LIN {X 0,Y 323.143,Z 396.929,A -85,B 0,C 180,E1 -15592.369,E2 -15592.369} C_VEL
LIN {X 0,Y 324.214,Z 384.488,A -85,B 0,C 180,E1 -15593.048,E2 -15593.048} C_VEL
LIN {X 0,Y 325.12,Z 370.663,A -85,B 0,C 180,E1 -15593.528,E2 -15593.528} C_VEL
LIN {X 0,Y 327.107,Z 306.154,A -85,B 0,C 180,E1 -15595.157,E2 -15595.157} C_VEL
LIN {X 0,Y 324.289,Z 289.299,A -85,B 0,C 180,E1 -15595.94,E2 -15595.94} C_VEL
LIN {X 0,Y 321.58,Z 277.548,A -85,B 0,C 180,E1 -15596.587,E2 -15596.587} C_VEL
LIN {X 0,Y 317.102,Z 267.049,A -85,B 0,C 180,E1 -15597.471,E2 -15597.471} C_VEL
LIN {X 0,Y 314.783,Z 256.674,A -85,B 0,C 180,E1 -15600.895,E2 -15600.895} C_VEL
LIN {X 0,Y 312.586,Z 248.4,A -85,B 0,C 180,E1 -15603.879,E2 -15603.879} C_VEL
LIN {X 0,Y 312.52,Z 248.065,A -85,B 0,C 180,E1 -15604.205,E2 -15604.205} C_VEL
LIN {X 0,Y 312.522,Z 248.055,A -85,B 0,C 180,E1 -15607.382,E2 -15607.382} C_VEL
LIN {X 0,Y 312.451,Z 248.063,A -85,B 0,C 180,E1 -15610.712,E2 -15610.712} C_VEL
LIN {X 0,Y 312.459,Z 248.066,A -85,B 0,C 180,E1 -15614.204,E2 -15614.204} C_VEL
LIN {X 0,Y 312.461,Z 248.06,A -85,B 0,C 180,E1 -15617.919,E2 -15617.919} C_VEL
LIN {X 0,Y 312.481,Z 248.06,A -85,B 0,C 180,E1 -15621.918,E2 -15621.918} C_VEL
LIN {X 0,Y 312.534,Z 248.049,A -85,B 0,C 180,E1 -15624.213,E2 -15624.213} C_VEL
LIN {X 0,Y 312.505,Z 248.053,A -85,B 0,C 180,E1 -15627.326,E2 -15627.326} C_VEL
LIN {X 0,Y 312.5,Z 248.058,A -85,B 0,C 180,E1 -15631.288,E2 -15631.288} C_VEL
LIN {X 0,Y 312.547,Z 248.049,A -85,B 0,C 180,E1 -15634.7,E2 -15634.7} C_VEL
LIN {X 0,Y 312.538,Z 248.046,A -85,B 0,C 180,E1 -15637.518,E2 -15637.518} C_VEL
LIN {X 0,Y 312.536,Z 248.051,A -85,B 0,C 180,E1 -15641.643,E2 -15641.643} C_VEL
LIN {X 0,Y 312.645,Z 248.04,A -85,B 0,C 180,E1 -15645.676,E2 -15645.676} C_VEL
LIN {X 0,Y 312.675,Z 248.037,A -85,B 0,C 180,E1 -15649.633,E2 -15649.633} C_VEL
LIN {X 0,Y 312.79,Z 248.021,A -85,B 0,C 180,E1 -15652.244,E2 -15652.244} C_VEL
LIN {X 0,Y 312.681,Z 248.031,A -85,B 0,C 180,E1 -15654.834,E2 -15654.834} C_VEL
LIN {X 0,Y 312.97,Z 248.001,A -85,B 0,C 180,E1 -15658.705,E2 -15658.705} C_VEL
LIN {X 0,Y 312.969,Z 248.002,A -85,B 0,C 180,E1 -15661.278,E2 -15661.278} C_VEL
LIN {X 0,Y 312.689,Z 248.033,A -85,B 0,C 180,E1 -15665.149,E2 -15665.149} C_VEL
LIN {X 0,Y 312.839,Z 248.019,A -85,B 0,C 180,E1 -15667.737,E2 -15667.737} C_VEL
LIN {X 0,Y 312.646,Z 248.042,A -85,B 0,C 180,E1 -15671.663,E2 -15671.663} C_VEL
LIN {X 0,Y 312.692,Z 248.117,A -85,B 0,C 180,E1 -15674.304,E2 -15674.304} C_VEL
LIN {X 0,Y 313.537,Z 251.516,A -85,B 0,C 180,E1 -15675.594,E2 -15675.594} C_VEL
LIN {X 0,Y 315.675,Z 259.924,A -85,B 0,C 180,E1 -15678.403,E2 -15678.403} C_VEL
LIN {X 0,Y 322.231,Z 274.036,A -85,B 0,C 180,E1 -15679.641,E2 -15679.641} C_VEL
LIN {X 0,Y 324.868,Z 280.655,A -85,B 0,C 180,E1 -15680.127,E2 -15680.127} C_VEL
LIN {X 0,Y 327.477,Z 294.554,A -85,B 0,C 180,E1 -15680.804,E2 -15680.804} C_VEL
LIN {X 0,Y 324.906,Z 368.524,A -85,B 0,C 180,E1 -15682.683,E2 -15682.683} C_VEL
LIN {X 0,Y 323.933,Z 382.296,A -85,B 0,C 180,E1 -15683.282,E2 -15683.282} C_VEL
LIN {X 0,Y 322.856,Z 394.211,A -85,B 0,C 180,E1 -15684.043,E2 -15684.043} C_VEL
LIN {X 0,Y 321.445,Z 406.032,A -85,B 0,C 180,E1 -15685.052,E2 -15685.052} C_VEL
LIN {X 0,Y 319.906,Z 416.817,A -85,B 0,C 180,E1 -15686.228,E2 -15686.228} C_VEL
LIN {X 0,Y 318.283,Z 427.014,A -85,B 0,C 180,E1 -15687.615,E2 -15687.615} C_VEL
LIN {X 0,Y 316.651,Z 436.505,A -85,B 0,C 180,E1 -15689.216,E2 -15689.216} C_VEL
LIN {X 0,Y 315.049,Z 445.372,A -85,B 0,C 180,E1 -15691.091,E2 -15691.091} C_VEL
LIN {X 0,Y 313.552,Z 453.218,A -85,B 0,C 180,E1 -15693.171,E2 -15693.171} C_VEL
LIN {X 0,Y 312.402,Z 459.627,A -85,B 0,C 180,E1 -15695.387,E2 -15695.387} C_VEL
LIN {X 0,Y 311.579,Z 464.294,A -85,B 0,C 180,E1 -15697.504,E2 -15697.504} C_VEL
LIN {X 0,Y 310.961,Z 467.929,A -85,B 0,C 180,E1 -15699.791,E2 -15699.791} C_VEL
LIN {X 0,Y 310.639,Z 469.904,A -85,B 0,C 180,E1 -15701.707,E2 -15701.707} C_VEL
LIN {X 0,Y 310.454,Z 470.97,A -85,B 0,C 180,E1 -15703.584,E2 -15703.584} C_VEL
LIN {X 0,Y 310.354,Z 471.2,A -85,B 0,C 180,E1 -15705.416,E2 -15705.416} C_VEL
LIN {X 0,Y 310.336,Z 470.655,A -85,B 0,C 180,E1 -15707.208,E2 -15707.208} C_VEL
LIN {X 0,Y 310.409,Z 469.328,A -85,B 0,C 180,E1 -15708.963,E2 -15708.963} C_VEL
LIN {X 0,Y 310.647,Z 467.257,A -85,B 0,C 180,E1 -15710.697,E2 -15710.697} C_VEL
LIN {X 0,Y 310.884,Z 464.494,A -85,B 0,C 180,E1 -15712.387,E2 -15712.387} C_VEL
LIN {X 0,Y 311.332,Z 460.269,A -85,B 0,C 180,E1 -15714.337,E2 -15714.337} C_VEL
LIN {X 0,Y 311.974,Z 454.336,A -85,B 0,C 180,E1 -15716.44,E2 -15716.44} C_VEL
LIN {X 0,Y 312.718,Z 447.541,A -85,B 0,C 180,E1 -15718.348,E2 -15718.348} C_VEL
LIN {X 0,Y 313.675,Z 439.821,A -85,B 0,C 180,E1 -15720.101,E2 -15720.101} C_VEL
LIN {X 0,Y 314.849,Z 430.134,A -85,B 0,C 180,E1 -15721.868,E2 -15721.868} C_VEL
LIN {X 0,Y 316.135,Z 419.363,A -85,B 0,C 180,E1 -15723.441,E2 -15723.441} C_VEL
LIN {X 0,Y 317.364,Z 407.822,A -85,B 0,C 180,E1 -15724.771,E2 -15724.771} C_VEL
LIN {X 0,Y 318.552,Z 394.945,A -85,B 0,C 180,E1 -15725.914,E2 -15725.914} C_VEL
LIN {X 0,Y 319.425,Z 382.214,A -85,B 0,C 180,E1 -15726.748,E2 -15726.748} C_VEL
LIN {X 0,Y 320.216,Z 368.151,A -85,B 0,C 180,E1 -15727.364,E2 -15727.364} C_VEL
LIN {X 0,Y 322.173,Z 291.979,A -85,B 0,C 180,E1 -15729.253,E2 -15729.253} C_VEL
LIN {X 0,Y 318.072,Z 269.596,A -85,B 0,C 180,E1 -15730.109,E2 -15730.109} C_VEL
LIN {X 0,Y 315.028,Z 260.599,A -85,B 0,C 180,E1 -15730.579,E2 -15730.579} C_VEL
LIN {X 0,Y 314.615,Z 258.571,A -85,B 0,C 180,E1 -15731.103,E2 -15731.103} C_VEL
LIN {X 0,Y 312.6,Z 248.111,A -85,B 0,C 180,E1 -15734.656,E2 -15734.656} C_VEL
LIN {X 0,Y 312.602,Z 248.047,A -85,B 0,C 180,E1 -15738.329,E2 -15738.329} C_VEL
LIN {X 0,Y 312.792,Z 248.021,A -85,B 0,C 180,E1 -15742.255,E2 -15742.255} C_VEL
LIN {X 0,Y 312.655,Z 248.041,A -85,B 0,C 180,E1 -15744.844,E2 -15744.844} C_VEL
LIN {X 0,Y 312.892,Z 248.008,A -85,B 0,C 180,E1 -15747.427,E2 -15747.427} C_VEL
LIN {X 0,Y 313.034,Z 247.988,A -85,B 0,C 180,E1 -15750.002,E2 -15750.002} C_VEL
LIN {X 0,Y 312.893,Z 248.008,A -85,B 0,C 180,E1 -15752.577,E2 -15752.577} C_VEL
LIN {X 0,Y 312.838,Z 248.013,A -85,B 0,C 180,E1 -15756.452,E2 -15756.452} C_VEL
LIN {X 0,Y 312.721,Z 248.031,A -85,B 0,C 180,E1 -15759.053,E2 -15759.053} C_VEL
LIN {X 0,Y 312.57,Z 248.048,A -85,B 0,C 180,E1 -15762.996,E2 -15762.996} C_VEL
LIN {X 0,Y 312.564,Z 248.051,A -85,B 0,C 180,E1 -15765.656,E2 -15765.656} C_VEL
LIN {X 0,Y 312.549,Z 248.047,A -85,B 0,C 180,E1 -15769.23,E2 -15769.23} C_VEL
LIN {X 0,Y 312.47,Z 248.059,A -85,B 0,C 180,E1 -15772.787,E2 -15772.787} C_VEL
LIN {X 0,Y 312.547,Z 248.052,A -85,B 0,C 180,E1 -15775.942,E2 -15775.942} C_VEL
LIN {X 0,Y 312.493,Z 248.051,A -85,B 0,C 180,E1 -15779.657,E2 -15779.657} C_VEL
LIN {X 0,Y 312.471,Z 248.06,A -85,B 0,C 180,E1 -15783.697,E2 -15783.697} C_VEL
LIN {X 0,Y 312.494,Z 248.055,A -85,B 0,C 180,E1 -15787.392,E2 -15787.392} C_VEL
LIN {X 0,Y 312.485,Z 248.06,A -85,B 0,C 180,E1 -15790.712,E2 -15790.712} C_VEL
LIN {X 0,Y 312.556,Z 248.051,A -85,B 0,C 180,E1 -15794.193,E2 -15794.193} C_VEL
LIN {X 0,Y 312.525,Z 248.049,A -85,B 0,C 180,E1 -15794.965,E2 -15794.965} C_VEL
LIN {X 0,Y 311.856,Z 248.137,A -85,B 0,C 180,E1 -15796.041,E2 -15796.041} C_VEL
LIN {X 0,Y 308.981,Z 248.492,A -85,B 0,C 180,E1 -15797.79,E2 -15797.79} C_VEL
LIN {X 0,Y 306.546,Z 248.798,A -85,B 0,C 180,E1 -15799.209,E2 -15799.209} C_VEL
LIN {X 0,Y 305.509,Z 248.928,A -85,B 0,C 180,E1 -15800.309,E2 -15800.309} C_VEL
LIN {X 0,Y 305.43,Z 248.932,A -85,B 0,C 180,E1 -15800.681,E2 -15800.681} C_VEL
LIN {X 0,Y 305.474,Z 248.929,A -85,B 0,C 180,E1 -15803.636,E2 -15803.636} C_VEL
LIN {X 0,Y 305.439,Z 248.934,A -85,B 0,C 180,E1 -15806.493,E2 -15806.493} C_VEL
LIN {X 0,Y 305.435,Z 248.936,A -85,B 0,C 180,E1 -15809.6,E2 -15809.6} C_VEL
LIN {X 0,Y 305.476,Z 248.931,A -85,B 0,C 180,E1 -15812.616,E2 -15812.616} C_VEL
LIN {X 0,Y 305.488,Z 248.93,A -85,B 0,C 180,E1 -15815.548,E2 -15815.548} C_VEL
LIN {X 0,Y 305.471,Z 248.932,A -85,B 0,C 180,E1 -15819.822,E2 -15819.822} C_VEL
LIN {X 0,Y 305.543,Z 248.921,A -85,B 0,C 180,E1 -15823.987,E2 -15823.987} C_VEL
LIN {X 0,Y 305.582,Z 248.916,A -85,B 0,C 180,E1 -15826.714,E2 -15826.714} C_VEL
LIN {X 0,Y 305.753,Z 248.896,A -85,B 0,C 180,E1 -15831.271,E2 -15831.271} C_VEL
LIN {X 0,Y 305.788,Z 248.89,A -85,B 0,C 180,E1 -15833.41,E2 -15833.41} C_VEL
LIN {X 0,Y 305.866,Z 248.883,A -85,B 0,C 180,E1 -15837.375,E2 -15837.375} C_VEL
LIN {X 0,Y 305.923,Z 248.879,A -85,B 0,C 180,E1 -15840.009,E2 -15840.009} C_VEL
LIN {X 0,Y 305.862,Z 248.878,A -85,B 0,C 180,E1 -15842.642,E2 -15842.642} C_VEL
LIN {X 0,Y 305.798,Z 248.887,A -85,B 0,C 180,E1 -15846.607,E2 -15846.607} C_VEL
LIN {X 0,Y 305.708,Z 248.899,A -85,B 0,C 180,E1 -15849.269,E2 -15849.269} C_VEL
LIN {X 0,Y 305.602,Z 248.915,A -85,B 0,C 180,E1 -15853.303,E2 -15853.303} C_VEL
LIN {X 0,Y 305.569,Z 248.918,A -85,B 0,C 180,E1 -15856.029,E2 -15856.029} C_VEL
LIN {X 0,Y 305.502,Z 248.923,A -85,B 0,C 180,E1 -15860.194,E2 -15860.194} C_VEL
LIN {X 0,Y 305.509,Z 248.93,A -85,B 0,C 180,E1 -15863.045,E2 -15863.045} C_VEL
LIN {X 0,Y 305.49,Z 248.928,A -85,B 0,C 180,E1 -15866.201,E2 -15866.201} C_VEL
LIN {X 0,Y 305.458,Z 248.933,A -85,B 0,C 180,E1 -15869.034,E2 -15869.034} C_VEL
LIN {X 0,Y 305.461,Z 248.932,A -85,B 0,C 180,E1 -15871.958,E2 -15871.958} C_VEL
LIN {X 0,Y 305.487,Z 248.933,A -85,B 0,C 180,E1 -15875.118,E2 -15875.118} C_VEL
LIN {X 0,Y 305.46,Z 248.932,A -85,B 0,C 180,E1 -15878.529,E2 -15878.529} C_VEL
LIN {X 0,Y 305.405,Z 248.937,A -85,B 0,C 180,E1 -15882.573,E2 -15882.573} C_VEL
LIN {X 0,Y 305.408,Z 248.938,A -85,B 0,C 180,E1 -15886.339,E2 -15886.339} C_VEL
LIN {X 0,Y 305.418,Z 248.942,A -85,B 0,C 180,E1 -15889.884,E2 -15889.884} C_VEL
LIN {X 0,Y 305.487,Z 248.934,A -85,B 0,C 180,E1 -15893.639,E2 -15893.639} C_VEL
LIN {X 0,Y 305.492,Z 248.931,A -85,B 0,C 180,E1 -15896.484,E2 -15896.484} C_VEL
LIN {X 0,Y 305.517,Z 249.096,A -85,B 0,C 180,E1 -15898.924,E2 -15898.924} C_VEL
LIN {X 0,Y 307.752,Z 259.847,A -85,B 0,C 180,E1 -15902.453,E2 -15902.453} C_VEL
LIN {X 0,Y 309.311,Z 268.287,A -85,B 0,C 180,E1 -15905.027,E2 -15905.027} C_VEL
LIN {X 0,Y 310.261,Z 273.009,A -85,B 0,C 180,E1 -15905.272,E2 -15905.272} C_VEL
LIN {X 0,Y 315.347,Z 307.012,A -85,B 0,C 180,E1 -15906.527,E2 -15906.527} C_VEL
LIN {X 0,Y 313.49,Z 375.371,A -85,B 0,C 180,E1 -15908.245,E2 -15908.245} C_VEL
LIN {X 0,Y 312.701,Z 389.193,A -85,B 0,C 180,E1 -15908.836,E2 -15908.836} C_VEL
LIN {X 0,Y 311.73,Z 401.738,A -85,B 0,C 180,E1 -15909.63,E2 -15909.63} C_VEL
LIN {X 0,Y 310.555,Z 413.817,A -85,B 0,C 180,E1 -15910.67,E2 -15910.67} C_VEL
LIN {X 0,Y 309.233,Z 425.375,A -85,B 0,C 180,E1 -15911.959,E2 -15911.959} C_VEL
LIN {X 0,Y 308.113,Z 435.341,A -85,B 0,C 180,E1 -15913.354,E2 -15913.354} C_VEL
LIN {X 0,Y 306.849,Z 445.2,A -85,B 0,C 180,E1 -15915.066,E2 -15915.066} C_VEL
LIN {X 0,Y 305.701,Z 454.297,A -85,B 0,C 180,E1 -15917.045,E2 -15917.045} C_VEL
LIN {X 0,Y 304.831,Z 461.601,A -85,B 0,C 180,E1 -15919.033,E2 -15919.033} C_VEL
LIN {X 0,Y 304.321,Z 466.519,A -85,B 0,C 180,E1 -15920.695,E2 -15920.695} C_VEL
LIN {X 0,Y 303.879,Z 471.271,A -85,B 0,C 180,E1 -15922.69,E2 -15922.69} C_VEL
LIN {X 0,Y 303.663,Z 474.872,A -85,B 0,C 180,E1 -15924.686,E2 -15924.686} C_VEL
LIN {X 0,Y 303.6,Z 476.688,A -85,B 0,C 180,E1 -15926.016,E2 -15926.016} C_VEL
LIN {X 0,Y 303.592,Z 478.049,A -85,B 0,C 180,E1 -15927.344,E2 -15927.344} C_VEL
LIN {X 0,Y 303.54,Z 479.001,A -85,B 0,C 180,E1 -15928.671,E2 -15928.671} C_VEL
LIN {X 0,Y 303.547,Z 479.553,A -85,B 0,C 180,E1 -15929.998,E2 -15929.998} C_VEL
LIN {X 0,Y 303.539,Z 479.658,A -85,B 0,C 180,E1 -15931.324,E2 -15931.324} C_VEL
LIN {X 0,Y 303.592,Z 479.358,A -85,B 0,C 180,E1 -15932.651,E2 -15932.651} C_VEL
LIN {X 0,Y 303.606,Z 478.665,A -85,B 0,C 180,E1 -15933.98,E2 -15933.98} C_VEL
LIN {X 0,Y 303.718,Z 477.175,A -85,B 0,C 180,E1 -15935.676,E2 -15935.676} C_VEL
LIN {X 0,Y 304.09,Z 474.055,A -85,B 0,C 180,E1 -15937.968,E2 -15937.968} C_VEL
LIN {X 0,Y 304.709,Z 470.241,A -85,B 0,C 180,E1 -15939.959,E2 -15939.959} C_VEL
LIN {X 0,Y 305.562,Z 465.301,A -85,B 0,C 180,E1 -15941.944,E2 -15941.944} C_VEL
LIN {X 0,Y 306.698,Z 459.092,A -85,B 0,C 180,E1 -15943.92,E2 -15943.92} C_VEL
LIN {X 0,Y 308.341,Z 451.381,A -85,B 0,C 180,E1 -15945.871,E2 -15945.871} C_VEL
LIN {X 0,Y 310.033,Z 441.588,A -85,B 0,C 180,E1 -15947.851,E2 -15947.851} C_VEL
LIN {X 0,Y 311.728,Z 431.881,A -85,B 0,C 180,E1 -15949.421,E2 -15949.421} C_VEL
LIN {X 0,Y 313.597,Z 420.806,A -85,B 0,C 180,E1 -15950.838,E2 -15950.838} C_VEL
LIN {X 0,Y 315.366,Z 408.317,A -85,B 0,C 180,E1 -15952.087,E2 -15952.087} C_VEL
LIN {X 0,Y 316.922,Z 396.004,A -85,B 0,C 180,E1 -15953.005,E2 -15953.005} C_VEL
LIN {X 0,Y 318.017,Z 383.244,A -85,B 0,C 180,E1 -15953.696,E2 -15953.696} C_VEL
LIN {X 0,Y 318.88,Z 370.165,A -85,B 0,C 180,E1 -15954.146,E2 -15954.146} C_VEL
LIN {X 0,Y 320.97,Z 307.114,A -85,B 0,C 180,E1 -15955.769,E2 -15955.769} C_VEL
LIN {X 0,Y 318.251,Z 290.858,A -85,B 0,C 180,E1 -15956.562,E2 -15956.562} C_VEL
LIN {X 0,Y 316.086,Z 280.936,A -85,B 0,C 180,E1 -15957.114,E2 -15957.114} C_VEL
LIN {X 0,Y 311.207,Z 269.934,A -85,B 0,C 180,E1 -15958.066,E2 -15958.066} C_VEL
LIN {X 0,Y 309.962,Z 267.008,A -85,B 0,C 180,E1 -15958.344,E2 -15958.344} C_VEL
LIN {X 0,Y 307.674,Z 257.238,A -85,B 0,C 180,E1 -15961.69,E2 -15961.69} C_VEL
LIN {X 0,Y 305.505,Z 249.086,A -85,B 0,C 180,E1 -15964.816,E2 -15964.816} C_VEL
LIN {X 0,Y 305.446,Z 248.939,A -85,B 0,C 180,E1 -15968.519,E2 -15968.519} C_VEL
LIN {X 0,Y 305.444,Z 248.937,A -85,B 0,C 180,E1 -15972.575,E2 -15972.575} C_VEL
LIN {X 0,Y 305.428,Z 248.939,A -85,B 0,C 180,E1 -15976.337,E2 -15976.337} C_VEL
LIN {X 0,Y 305.417,Z 248.94,A -85,B 0,C 180,E1 -15979.878,E2 -15979.878} C_VEL
LIN {X 0,Y 305.466,Z 248.928,A -85,B 0,C 180,E1 -15983.631,E2 -15983.631} C_VEL
LIN {X 0,Y 305.469,Z 248.929,A -85,B 0,C 180,E1 -15986.476,E2 -15986.476} C_VEL
LIN {X 0,Y 305.421,Z 248.936,A -85,B 0,C 180,E1 -15989.579,E2 -15989.579} C_VEL
LIN {X 0,Y 305.455,Z 248.933,A -85,B 0,C 180,E1 -15992.594,E2 -15992.594} C_VEL
LIN {X 0,Y 305.473,Z 248.933,A -85,B 0,C 180,E1 -15995.528,E2 -15995.528} C_VEL
LIN {X 0,Y 305.456,Z 248.933,A -85,B 0,C 180,E1 -15998.392,E2 -15998.392} C_VEL
LIN {X 0,Y 305.495,Z 248.924,A -85,B 0,C 180,E1 -16001.204,E2 -16001.204} C_VEL
LIN {X 0,Y 305.572,Z 248.919,A -85,B 0,C 180,E1 -16005.337,E2 -16005.337} C_VEL
LIN {X 0,Y 305.614,Z 248.918,A -85,B 0,C 180,E1 -16009.391,E2 -16009.391} C_VEL
LIN {X 0,Y 305.74,Z 248.899,A -85,B 0,C 180,E1 -16012.064,E2 -16012.064} C_VEL
LIN {X 0,Y 305.651,Z 248.906,A -85,B 0,C 180,E1 -16014.714,E2 -16014.714} C_VEL
LIN {X 0,Y 305.936,Z 248.877,A -85,B 0,C 180,E1 -16018.675,E2 -16018.675} C_VEL
LIN {X 0,Y 305.936,Z 248.879,A -85,B 0,C 180,E1 -16021.308,E2 -16021.308} C_VEL
LIN {X 0,Y 305.661,Z 248.909,A -85,B 0,C 180,E1 -16025.268,E2 -16025.268} C_VEL
LIN {X 0,Y 305.782,Z 248.898,A -85,B 0,C 180,E1 -16027.917,E2 -16027.917} C_VEL
LIN {X 0,Y 305.58,Z 248.921,A -85,B 0,C 180,E1 -16031.936,E2 -16031.936} C_VEL
LIN {X 0,Y 305.601,Z 248.982,A -85,B 0,C 180,E1 -16033.455,E2 -16033.455} C_VEL
LIN {X 0,Y 307.131,Z 254.679,A -85,B 0,C 180,E1 -16035.653,E2 -16035.653} C_VEL
LIN {X 0,Y 308.543,Z 260.196,A -85,B 0,C 180,E1 -16037.522,E2 -16037.522} C_VEL
LIN {X 0,Y 314.968,Z 273.498,A -85,B 0,C 180,E1 -16038.783,E2 -16038.783} C_VEL
LIN {X 0,Y 319.191,Z 283.718,A -85,B 0,C 180,E1 -16039.588,E2 -16039.588} C_VEL
LIN {X 0,Y 321.366,Z 295.811,A -85,B 0,C 180,E1 -16040.196,E2 -16040.196} C_VEL
LIN {X 0,Y 318.671,Z 368.497,A -85,B 0,C 180,E1 -16042.078,E2 -16042.078} C_VEL
LIN {X 0,Y 317.615,Z 382.644,A -85,B 0,C 180,E1 -16042.703,E2 -16042.703} C_VEL
LIN {X 0,Y 316.41,Z 395.453,A -85,B 0,C 180,E1 -16043.555,E2 -16043.555} C_VEL
LIN {X 0,Y 314.75,Z 408.209,A -85,B 0,C 180,E1 -16044.699,E2 -16044.699} C_VEL
LIN {X 0,Y 313.273,Z 417.956,A -85,B 0,C 180,E1 -16045.816,E2 -16045.816} C_VEL
LIN {X 0,Y 311.448,Z 428.762,A -85,B 0,C 180,E1 -16047.361,E2 -16047.361} C_VEL
LIN {X 0,Y 309.732,Z 437.936,A -85,B 0,C 180,E1 -16049.001,E2 -16049.001} C_VEL
LIN {X 0,Y 308.111,Z 446.353,A -85,B 0,C 180,E1 -16050.866,E2 -16050.866} C_VEL
LIN {X 0,Y 306.525,Z 454.18,A -85,B 0,C 180,E1 -16053.056,E2 -16053.056} C_VEL
LIN {X 0,Y 305.429,Z 459.882,A -85,B 0,C 180,E1 -16055.104,E2 -16055.104} C_VEL
LIN {X 0,Y 304.475,Z 465.022,A -85,B 0,C 180,E1 -16057.538,E2 -16057.538} C_VEL
LIN {X 0,Y 303.964,Z 467.842,A -85,B 0,C 180,E1 -16059.404,E2 -16059.404} C_VEL
LIN {X 0,Y 303.745,Z 468.961,A -85,B 0,C 180,E1 -16060.366,E2 -16060.366} C_VEL
LIN {X 0,Y 303.483,Z 470.477,A -85,B 0,C 180,E1 -16062.183,E2 -16062.183} C_VEL
LIN {X 0,Y 303.309,Z 471.256,A -85,B 0,C 180,E1 -16064.089,E2 -16064.089} C_VEL
LIN {X 0,Y 303.256,Z 471.21,A -85,B 0,C 180,E1 -16065.956,E2 -16065.956} C_VEL
LIN {X 0,Y 303.261,Z 470.311,A -85,B 0,C 180,E1 -16067.85,E2 -16067.85} C_VEL
LIN {X 0,Y 303.404,Z 468.473,A -85,B 0,C 180,E1 -16069.836,E2 -16069.836} C_VEL
LIN {X 0,Y 303.728,Z 465.6,A -85,B 0,C 180,E1 -16071.862,E2 -16071.862} C_VEL
LIN {X 0,Y 304.141,Z 461.488,A -85,B 0,C 180,E1 -16073.955,E2 -16073.955} C_VEL
LIN {X 0,Y 304.736,Z 455.931,A -85,B 0,C 180,E1 -16076.103,E2 -16076.103} C_VEL
LIN {X 0,Y 305.6,Z 448.588,A -85,B 0,C 180,E1 -16078.287,E2 -16078.287} C_VEL
LIN {X 0,Y 306.581,Z 440.79,A -85,B 0,C 180,E1 -16080.14,E2 -16080.14} C_VEL
LIN {X 0,Y 307.725,Z 431.805,A -85,B 0,C 180,E1 -16081.872,E2 -16081.872} C_VEL
LIN {X 0,Y 309.047,Z 421.239,A -85,B 0,C 180,E1 -16083.497,E2 -16083.497} C_VEL
LIN {X 0,Y 310.332,Z 409.706,A -85,B 0,C 180,E1 -16084.912,E2 -16084.912} C_VEL
LIN {X 0,Y 311.477,Z 397.841,A -85,B 0,C 180,E1 -16086.04,E2 -16086.04} C_VEL
LIN {X 0,Y 312.437,Z 385.507,A -85,B 0,C 180,E1 -16086.928,E2 -16086.928} C_VEL
LIN {X 0,Y 313.255,Z 372.677,A -85,B 0,C 180,E1 -16087.582,E2 -16087.582} C_VEL
LIN {X 0,Y 313.807,Z 357.919,A -85,B 0,C 180,E1 -16088.035,E2 -16088.035} C_VEL
LIN {X 0,Y 315.483,Z 292.998,A -85,B 0,C 180,E1 -16089.654,E2 -16089.654} C_VEL
LIN {X 0,Y 311.694,Z 271.957,A -85,B 0,C 180,E1 -16090.47,E2 -16090.47} C_VEL
LIN {X 0,Y 307.771,Z 260.477,A -85,B 0,C 180,E1 -16091.099,E2 -16091.099} C_VEL
LIN {X 0,Y 306.433,Z 253.556,A -85,B 0,C 180,E1 -16093.343,E2 -16093.343} C_VEL
LIN {X 0,Y 305.603,Z 248.978,A -85,B 0,C 180,E1 -16094.993,E2 -16094.993} C_VEL
LIN {X 0,Y 305.57,Z 248.92,A -85,B 0,C 180,E1 -16099.4,E2 -16099.4} C_VEL
LIN {X 0,Y 305.734,Z 248.899,A -85,B 0,C 180,E1 -16102.075,E2 -16102.075} C_VEL
LIN {X 0,Y 305.625,Z 248.917,A -85,B 0,C 180,E1 -16104.725,E2 -16104.725} C_VEL
LIN {X 0,Y 305.894,Z 248.882,A -85,B 0,C 180,E1 -16108.686,E2 -16108.686} C_VEL
LIN {X 0,Y 305.895,Z 248.882,A -85,B 0,C 180,E1 -16111.319,E2 -16111.319} C_VEL
LIN {X 0,Y 305.627,Z 248.916,A -85,B 0,C 180,E1 -16115.28,E2 -16115.28} C_VEL
LIN {X 0,Y 305.738,Z 248.898,A -85,B 0,C 180,E1 -16117.93,E2 -16117.93} C_VEL
LIN {X 0,Y 305.54,Z 248.923,A -85,B 0,C 180,E1 -16121.95,E2 -16121.95} C_VEL
LIN {X 0,Y 305.558,Z 248.922,A -85,B 0,C 180,E1 -16125.027,E2 -16125.027} C_VEL
LIN {X 0,Y 305.519,Z 248.92,A -85,B 0,C 180,E1 -16128.789,E2 -16128.789} C_VEL
LIN {X 0,Y 305.43,Z 248.936,A -85,B 0,C 180,E1 -16133.046,E2 -16133.046} C_VEL
LIN {X 0,Y 305.477,Z 248.929,A -85,B 0,C 180,E1 -16136.228,E2 -16136.228} C_VEL
LIN {X 0,Y 305.442,Z 248.926,A -85,B 0,C 180,E1 -16139.057,E2 -16139.057} C_VEL
LIN {X 0,Y 305.397,Z 248.941,A -85,B 0,C 180,E1 -16141.96,E2 -16141.96} C_VEL
LIN {X 0,Y 305.414,Z 248.938,A -85,B 0,C 180,E1 -16145.122,E2 -16145.122} C_VEL
LIN {X 0,Y 305.438,Z 248.937,A -85,B 0,C 180,E1 -16148.545,E2 -16148.545} C_VEL
LIN {X 0,Y 305.481,Z 248.934,A -85,B 0,C 180,E1 -16152.608,E2 -16152.608} C_VEL
LIN {X 0,Y 305.497,Z 248.93,A -85,B 0,C 180,E1 -16156.374,E2 -16156.374} C_VEL
LIN {X 0,Y 305.453,Z 248.933,A -85,B 0,C 180,E1 -16159.906,E2 -16159.906} C_VEL
LIN {X 0,Y 305.43,Z 248.932,A -85,B 0,C 180,E1 -16160.681,E2 -16160.681} C_VEL
LIN {X 0,Y 304.768,Z 249.019,A -85,B 0,C 180,E1 -16161.781,E2 -16161.781} C_VEL
LIN {X 0,Y 301.899,Z 249.374,A -85,B 0,C 180,E1 -16163.572,E2 -16163.572} C_VEL
LIN {X 0,Y 299.464,Z 249.68,A -85,B 0,C 180,E1 -16165.025,E2 -16165.025} C_VEL
LIN {X 0,Y 298.426,Z 249.805,A -85,B 0,C 180,E1 -16166.15,E2 -16166.15} C_VEL
LIN {X 0,Y 298.346,Z 249.815,A -85,B 0,C 180,E1 -16166.532,E2 -16166.532} C_VEL
LIN {X 0,Y 298.406,Z 249.813,A -85,B 0,C 180,E1 -16170.627,E2 -16170.627} C_VEL
LIN {X 0,Y 298.458,Z 249.803,A -85,B 0,C 180,E1 -16173.488,E2 -16173.488} C_VEL
LIN {X 0,Y 298.416,Z 249.809,A -85,B 0,C 180,E1 -16176.71,E2 -16176.71} C_VEL
LIN {X 0,Y 298.453,Z 249.805,A -85,B 0,C 180,E1 -16180.762,E2 -16180.762} C_VEL
LIN {X 0,Y 298.58,Z 249.787,A -85,B 0,C 180,E1 -16185.004,E2 -16185.004} C_VEL
LIN {X 0,Y 298.589,Z 249.789,A -85,B 0,C 180,E1 -16189.156,E2 -16189.156} C_VEL
LIN {X 0,Y 298.699,Z 249.775,A -85,B 0,C 180,E1 -16191.894,E2 -16191.894} C_VEL
LIN {X 0,Y 298.636,Z 249.781,A -85,B 0,C 180,E1 -16194.608,E2 -16194.608} C_VEL
LIN {X 0,Y 298.91,Z 249.748,A -85,B 0,C 180,E1 -16198.662,E2 -16198.662} C_VEL
LIN {X 0,Y 298.92,Z 249.744,A -85,B 0,C 180,E1 -16201.356,E2 -16201.356} C_VEL
LIN {X 0,Y 298.746,Z 249.763,A -85,B 0,C 180,E1 -16206.763,E2 -16206.763} C_VEL
LIN {X 0,Y 298.639,Z 249.78,A -85,B 0,C 180,E1 -16209.49,E2 -16209.49} C_VEL
LIN {X 0,Y 298.562,Z 249.792,A -85,B 0,C 180,E1 -16213.623,E2 -16213.623} C_VEL
LIN {X 0,Y 298.502,Z 249.801,A -85,B 0,C 180,E1 -16216.419,E2 -16216.419} C_VEL
LIN {X 0,Y 298.465,Z 249.798,A -85,B 0,C 180,E1 -16219.625,E2 -16219.625} C_VEL
LIN {X 0,Y 298.442,Z 249.807,A -85,B 0,C 180,E1 -16223.607,E2 -16223.607} C_VEL
LIN {X 0,Y 298.43,Z 249.81,A -85,B 0,C 180,E1 -16226.588,E2 -16226.588} C_VEL
LIN {X 0,Y 298.385,Z 249.812,A -85,B 0,C 180,E1 -16229.653,E2 -16229.653} C_VEL
LIN {X 0,Y 298.418,Z 249.812,A -85,B 0,C 180,E1 -16232.805,E2 -16232.805} C_VEL
LIN {X 0,Y 298.429,Z 249.804,A -85,B 0,C 180,E1 -16236.076,E2 -16236.076} C_VEL
LIN {X 0,Y 298.399,Z 249.817,A -85,B 0,C 180,E1 -16239.496,E2 -16239.496} C_VEL
LIN {X 0,Y 298.367,Z 249.815,A -85,B 0,C 180,E1 -16243.094,E2 -16243.094} C_VEL
LIN {X 0,Y 298.367,Z 249.814,A -85,B 0,C 180,E1 -16246.912,E2 -16246.912} C_VEL
LIN {X 0,Y 298.389,Z 249.814,A -85,B 0,C 180,E1 -16251.019,E2 -16251.019} C_VEL
LIN {X 0,Y 298.43,Z 249.813,A -85,B 0,C 180,E1 -16253.93,E2 -16253.93} C_VEL
LIN {X 0,Y 298.42,Z 249.812,A -85,B 0,C 180,E1 -16257.201,E2 -16257.201} C_VEL
LIN {X 0,Y 298.466,Z 250.004,A -85,B 0,C 180,E1 -16258.583,E2 -16258.583} C_VEL
LIN {X 0,Y 300.654,Z 260.561,A -85,B 0,C 180,E1 -16262.125,E2 -16262.125} C_VEL
LIN {X 0,Y 302.165,Z 268.328,A -85,B 0,C 180,E1 -16264.541,E2 -16264.541} C_VEL
LIN {X 0,Y 303.685,Z 274.375,A -85,B 0,C 180,E1 -16264.856,E2 -16264.856} C_VEL
LIN {X 0,Y 308.657,Z 307.144,A -85,B 0,C 180,E1 -16266.102,E2 -16266.102} C_VEL
LIN {X 0,Y 306.701,Z 375.684,A -85,B 0,C 180,E1 -16267.871,E2 -16267.871} C_VEL
LIN {X 0,Y 305.879,Z 389.329,A -85,B 0,C 180,E1 -16268.473,E2 -16268.473} C_VEL
LIN {X 0,Y 304.848,Z 402.357,A -85,B 0,C 180,E1 -16269.326,E2 -16269.326} C_VEL
LIN {X 0,Y 303.639,Z 414.234,A -85,B 0,C 180,E1 -16270.388,E2 -16270.388} C_VEL
LIN {X 0,Y 302.281,Z 425.7,A -85,B 0,C 180,E1 -16271.705,E2 -16271.705} C_VEL
LIN {X 0,Y 301.151,Z 435.516,A -85,B 0,C 180,E1 -16273.119,E2 -16273.119} C_VEL
LIN {X 0,Y 299.968,Z 444.552,A -85,B 0,C 180,E1 -16274.715,E2 -16274.715} C_VEL
LIN {X 0,Y 298.753,Z 453.743,A -85,B 0,C 180,E1 -16276.738,E2 -16276.738} C_VEL
LIN {X 0,Y 297.825,Z 461.137,A -85,B 0,C 180,E1 -16278.772,E2 -16278.772} C_VEL
LIN {X 0,Y 297.286,Z 466.118,A -85,B 0,C 180,E1 -16280.472,E2 -16280.472} C_VEL
LIN {X 0,Y 296.828,Z 470.936,A -85,B 0,C 180,E1 -16282.515,E2 -16282.515} C_VEL
LIN {X 0,Y 296.578,Z 474.597,A -85,B 0,C 180,E1 -16284.559,E2 -16284.559} C_VEL
LIN {X 0,Y 296.504,Z 476.467,A -85,B 0,C 180,E1 -16285.92,E2 -16285.92} C_VEL
LIN {X 0,Y 296.497,Z 477.856,A -85,B 0,C 180,E1 -16287.28,E2 -16287.28} C_VEL
LIN {X 0,Y 296.463,Z 478.836,A -85,B 0,C 180,E1 -16288.639,E2 -16288.639} C_VEL
LIN {X 0,Y 296.465,Z 479.417,A -85,B 0,C 180,E1 -16289.998,E2 -16289.998} C_VEL
LIN {X 0,Y 296.461,Z 479.571,A -85,B 0,C 180,E1 -16291.356,E2 -16291.356} C_VEL
LIN {X 0,Y 296.498,Z 479.296,A -85,B 0,C 180,E1 -16292.715,E2 -16292.715} C_VEL
LIN {X 0,Y 296.509,Z 478.628,A -85,B 0,C 180,E1 -16294.075,E2 -16294.075} C_VEL
LIN {X 0,Y 296.604,Z 477.441,A -85,B 0,C 180,E1 -16295.574,E2 -16295.574} C_VEL
LIN {X 0,Y 297.058,Z 474.116,A -85,B 0,C 180,E1 -16298.158,E2 -16298.158} C_VEL
LIN {X 0,Y 297.704,Z 470.353,A -85,B 0,C 180,E1 -16300.196,E2 -16300.196} C_VEL
LIN {X 0,Y 298.614,Z 465.482,A -85,B 0,C 180,E1 -16302.226,E2 -16302.226} C_VEL
LIN {X 0,Y 299.82,Z 459.358,A -85,B 0,C 180,E1 -16304.246,E2 -16304.246} C_VEL
LIN {X 0,Y 301.536,Z 451.753,A -85,B 0,C 180,E1 -16306.239,E2 -16306.239} C_VEL
LIN {X 0,Y 303.128,Z 443.106,A -85,B 0,C 180,E1 -16308.072,E2 -16308.072} C_VEL
LIN {X 0,Y 304.876,Z 433.559,A -85,B 0,C 180,E1 -16309.7,E2 -16309.7} C_VEL
LIN {X 0,Y 306.763,Z 422.953,A -85,B 0,C 180,E1 -16311.149,E2 -16311.149} C_VEL
LIN {X 0,Y 308.392,Z 412.764,A -85,B 0,C 180,E1 -16312.261,E2 -16312.261} C_VEL
LIN {X 0,Y 310.127,Z 400.734,A -85,B 0,C 180,E1 -16313.273,E2 -16313.273} C_VEL
LIN {X 0,Y 311.389,Z 387.754,A -85,B 0,C 180,E1 -16314.1,E2 -16314.1} C_VEL
LIN {X 0,Y 312.449,Z 375.125,A -85,B 0,C 180,E1 -16314.632,E2 -16314.632} C_VEL
LIN {X 0,Y 314.907,Z 308.047,A -85,B 0,C 180,E1 -16316.417,E2 -16316.417} C_VEL
LIN {X 0,Y 312.328,Z 292.521,A -85,B 0,C 180,E1 -16317.202,E2 -16317.202} C_VEL
LIN {X 0,Y 310.387,Z 283.805,A -85,B 0,C 180,E1 -16317.715,E2 -16317.715} C_VEL
LIN {X 0,Y 304.742,Z 270.974,A -85,B 0,C 180,E1 -16318.873,E2 -16318.873} C_VEL
LIN {X 0,Y 302.669,Z 266.657,A -85,B 0,C 180,E1 -16319.355,E2 -16319.355} C_VEL
LIN {X 0,Y 300.513,Z 257.553,A -85,B 0,C 180,E1 -16322.647,E2 -16322.647} C_VEL
LIN {X 0,Y 298.439,Z 249.914,A -85,B 0,C 180,E1 -16325.753,E2 -16325.753} C_VEL
LIN {X 0,Y 298.386,Z 249.815,A -85,B 0,C 180,E1 -16329.486,E2 -16329.486} C_VEL
LIN {X 0,Y 298.379,Z 249.814,A -85,B 0,C 180,E1 -16333.09,E2 -16333.09} C_VEL
LIN {X 0,Y 298.378,Z 249.818,A -85,B 0,C 180,E1 -16336.908,E2 -16336.908} C_VEL
LIN {X 0,Y 298.392,Z 249.811,A -85,B 0,C 180,E1 -16341.004,E2 -16341.004} C_VEL
LIN {X 0,Y 298.408,Z 249.808,A -85,B 0,C 180,E1 -16343.921,E2 -16343.921} C_VEL
LIN {X 0,Y 298.397,Z 249.809,A -85,B 0,C 180,E1 -16347.192,E2 -16347.192} C_VEL
LIN {X 0,Y 298.373,Z 249.812,A -85,B 0,C 180,E1 -16350.629,E2 -16350.629} C_VEL
LIN {X 0,Y 298.438,Z 249.809,A -85,B 0,C 180,E1 -16354.912,E2 -16354.912} C_VEL
LIN {X 0,Y 298.396,Z 249.809,A -85,B 0,C 180,E1 -16357.854,E2 -16357.854} C_VEL
LIN {X 0,Y 298.448,Z 249.801,A -85,B 0,C 180,E1 -16360.743,E2 -16360.743} C_VEL
LIN {X 0,Y 298.505,Z 249.796,A -85,B 0,C 180,E1 -16364.982,E2 -16364.982} C_VEL
LIN {X 0,Y 298.573,Z 249.793,A -85,B 0,C 180,E1 -16369.138,E2 -16369.138} C_VEL
LIN {X 0,Y 298.691,Z 249.775,A -85,B 0,C 180,E1 -16371.876,E2 -16371.876} C_VEL
LIN {X 0,Y 298.621,Z 249.781,A -85,B 0,C 180,E1 -16374.59,E2 -16374.59} C_VEL
LIN {X 0,Y 298.902,Z 249.753,A -85,B 0,C 180,E1 -16378.644,E2 -16378.644} C_VEL
LIN {X 0,Y 298.903,Z 249.755,A -85,B 0,C 180,E1 -16381.338,E2 -16381.338} C_VEL
LIN {X 0,Y 298.765,Z 249.768,A -85,B 0,C 180,E1 -16386.745,E2 -16386.745} C_VEL
LIN {X 0,Y 298.657,Z 249.784,A -85,B 0,C 180,E1 -16389.472,E2 -16389.472} C_VEL
LIN {X 0,Y 298.539,Z 249.892,A -85,B 0,C 180,E1 -16392.567,E2 -16392.567} C_VEL
LIN {X 0,Y 299.669,Z 253.937,A -85,B 0,C 180,E1 -16394.246,E2 -16394.246} C_VEL
LIN {X 0,Y 301.373,Z 260.337,A -85,B 0,C 180,E1 -16396.548,E2 -16396.548} C_VEL
LIN {X 0,Y 307.944,Z 273.448,A -85,B 0,C 180,E1 -16397.896,E2 -16397.896} C_VEL
LIN {X 0,Y 313.33,Z 285.865,A -85,B 0,C 180,E1 -16398.97,E2 -16398.97} C_VEL
LIN {X 0,Y 315.274,Z 296.434,A -85,B 0,C 180,E1 -16399.524,E2 -16399.524} C_VEL
LIN {X 0,Y 312.476,Z 368.943,A -85,B 0,C 180,E1 -16401.459,E2 -16401.459} C_VEL
LIN {X 0,Y 311.348,Z 383.161,A -85,B 0,C 180,E1 -16402.107,E2 -16402.107} C_VEL
LIN {X 0,Y 310.139,Z 395.068,A -85,B 0,C 180,E1 -16402.911,E2 -16402.911} C_VEL
LIN {X 0,Y 308.402,Z 408.041,A -85,B 0,C 180,E1 -16404.09,E2 -16404.09} C_VEL
LIN {X 0,Y 306.558,Z 419.558,A -85,B 0,C 180,E1 -16405.447,E2 -16405.447} C_VEL
LIN {X 0,Y 304.737,Z 429.822,A -85,B 0,C 180,E1 -16406.989,E2 -16406.989} C_VEL
LIN {X 0,Y 302.913,Z 438.955,A -85,B 0,C 180,E1 -16408.684,E2 -16408.684} C_VEL
LIN {X 0,Y 301.409,Z 446.379,A -85,B 0,C 180,E1 -16410.381,E2 -16410.381} C_VEL
LIN {X 0,Y 299.786,Z 453.706,A -85,B 0,C 180,E1 -16412.445,E2 -16412.445} C_VEL
LIN {X 0,Y 298.607,Z 459.518,A -85,B 0,C 180,E1 -16414.542,E2 -16414.542} C_VEL
LIN {X 0,Y 297.704,Z 464.001,A -85,B 0,C 180,E1 -16416.621,E2 -16416.621} C_VEL
LIN {X 0,Y 297.044,Z 467.329,A -85,B 0,C 180,E1 -16418.673,E2 -16418.673} C_VEL
LIN {X 0,Y 296.596,Z 469.618,A -85,B 0,C 180,E1 -16420.694,E2 -16420.694} C_VEL
LIN {X 0,Y 296.332,Z 470.972,A -85,B 0,C 180,E1 -16422.679,E2 -16422.679} C_VEL
LIN {X 0,Y 296.159,Z 471.377,A -85,B 0,C 180,E1 -16425.374,E2 -16425.374} C_VEL
LIN {X 0,Y 296.143,Z 470.679,A -85,B 0,C 180,E1 -16427.348,E2 -16427.348} C_VEL
LIN {X 0,Y 296.247,Z 469.063,A -85,B 0,C 180,E1 -16429.371,E2 -16429.371} C_VEL
LIN {X 0,Y 296.652,Z 465.552,A -85,B 0,C 180,E1 -16431.981,E2 -16431.981} C_VEL
LIN {X 0,Y 296.977,Z 462.234,A -85,B 0,C 180,E1 -16433.731,E2 -16433.731} C_VEL
LIN {X 0,Y 297.633,Z 456.394,A -85,B 0,C 180,E1 -16436.098,E2 -16436.098} C_VEL
LIN {X 0,Y 298.339,Z 450.46,A -85,B 0,C 180,E1 -16437.978,E2 -16437.978} C_VEL
LIN {X 0,Y 299.372,Z 442.687,A -85,B 0,C 180,E1 -16439.957,E2 -16439.957} C_VEL
LIN {X 0,Y 300.641,Z 432.935,A -85,B 0,C 180,E1 -16441.939,E2 -16441.939} C_VEL
LIN {X 0,Y 301.915,Z 422.932,A -85,B 0,C 180,E1 -16443.567,E2 -16443.567} C_VEL
LIN {X 0,Y 303.286,Z 411.364,A -85,B 0,C 180,E1 -16445.055,E2 -16445.055} C_VEL
LIN {X 0,Y 304.512,Z 399.323,A -85,B 0,C 180,E1 -16446.271,E2 -16446.271} C_VEL
LIN {X 0,Y 305.597,Z 386.18,A -85,B 0,C 180,E1 -16447.257,E2 -16447.257} C_VEL
LIN {X 0,Y 306.473,Z 372.639,A -85,B 0,C 180,E1 -16447.969,E2 -16447.969} C_VEL
LIN {X 0,Y 307.077,Z 356.867,A -85,B 0,C 180,E1 -16448.456,E2 -16448.456} C_VEL
LIN {X 0,Y 308.742,Z 293.497,A -85,B 0,C 180,E1 -16450.081,E2 -16450.081} C_VEL
LIN {X 0,Y 305.211,Z 274.1,A -85,B 0,C 180,E1 -16450.859,E2 -16450.859} C_VEL
LIN {X 0,Y 300.611,Z 260.65,A -85,B 0,C 180,E1 -16451.605,E2 -16451.605} C_VEL
LIN {X 0,Y 299.76,Z 256.418,A -85,B 0,C 180,E1 -16452.961,E2 -16452.961} C_VEL
LIN {X 0,Y 298.559,Z 249.843,A -85,B 0,C 180,E1 -16455.344,E2 -16455.344} C_VEL
LIN {X 0,Y 298.525,Z 249.799,A -85,B 0,C 180,E1 -16459.147,E2 -16459.147} C_VEL
LIN {X 0,Y 298.682,Z 249.777,A -85,B 0,C 180,E1 -16461.886,E2 -16461.886} C_VEL
LIN {X 0,Y 298.595,Z 249.792,A -85,B 0,C 180,E1 -16464.6,E2 -16464.6} C_VEL
LIN {X 0,Y 298.861,Z 249.758,A -85,B 0,C 180,E1 -16468.655,E2 -16468.655} C_VEL
LIN {X 0,Y 298.862,Z 249.758,A -85,B 0,C 180,E1 -16471.35,E2 -16471.35} C_VEL
LIN {X 0,Y 298.597,Z 249.791,A -85,B 0,C 180,E1 -16475.404,E2 -16475.404} C_VEL
LIN {X 0,Y 298.685,Z 249.776,A -85,B 0,C 180,E1 -16478.118,E2 -16478.118} C_VEL
LIN {X 0,Y 298.49,Z 249.8,A -85,B 0,C 180,E1 -16482.236,E2 -16482.236} C_VEL
LIN {X 0,Y 298.497,Z 249.802,A -85,B 0,C 180,E1 -16485.18,E2 -16485.18} C_VEL
LIN {X 0,Y 298.465,Z 249.8,A -85,B 0,C 180,E1 -16489.25,E2 -16489.25} C_VEL
LIN {X 0,Y 298.373,Z 249.819,A -85,B 0,C 180,E1 -16493.607,E2 -16493.607} C_VEL
LIN {X 0,Y 298.433,Z 249.804,A -85,B 0,C 180,E1 -16496.582,E2 -16496.582} C_VEL
LIN {X 0,Y 298.37,Z 249.807,A -85,B 0,C 180,E1 -16499.649,E2 -16499.649} C_VEL
LIN {X 0,Y 298.348,Z 249.818,A -85,B 0,C 180,E1 -16502.808,E2 -16502.808} C_VEL
LIN {X 0,Y 298.406,Z 249.811,A -85,B 0,C 180,E1 -16506.817,E2 -16506.817} C_VEL
LIN {X 0,Y 298.412,Z 249.81,A -85,B 0,C 180,E1 -16511.111,E2 -16511.111} C_VEL
LIN {X 0,Y 298.451,Z 249.805,A -85,B 0,C 180,E1 -16515.07,E2 -16515.07} C_VEL
LIN {X 0,Y 298.42,Z 249.812,A -85,B 0,C 180,E1 -16518.908,E2 -16518.908} C_VEL
LIN {X 0,Y 298.442,Z 249.807,A -85,B 0,C 180,E1 -16523.196,E2 -16523.196} C_VEL
LIN {X 0,Y 298.346,Z 249.815,A -85,B 0,C 180,E1 -16526.532,E2 -16526.532} C_VEL
LIN {X 0,Y 297.681,Z 249.903,A -85,B 0,C 180,E1 -16527.66,E2 -16527.66} C_VEL
LIN {X 0,Y 294.814,Z 250.26,A -85,B 0,C 180,E1 -16529.496,E2 -16529.496} C_VEL
LIN {X 0,Y 292.413,Z 250.562,A -85,B 0,C 180,E1 -16530.987,E2 -16530.987} C_VEL
LIN {X 0,Y 291.432,Z 250.679,A -85,B 0,C 180,E1 -16532.141,E2 -16532.141} C_VEL
LIN {X 0,Y 291.378,Z 250.686,A -85,B 0,C 180,E1 -16532.532,E2 -16532.532} C_VEL
LIN {X 0,Y 291.37,Z 250.685,A -85,B 0,C 180,E1 -16536.435,E2 -16536.435} C_VEL
LIN {X 0,Y 291.381,Z 250.686,A -85,B 0,C 180,E1 -16540.276,E2 -16540.276} C_VEL
LIN {X 0,Y 291.492,Z 250.668,A -85,B 0,C 180,E1 -16544.676,E2 -16544.676} C_VEL
LIN {X 0,Y 291.533,Z 250.667,A -85,B 0,C 180,E1 -16548.891,E2 -16548.891} C_VEL
LIN {X 0,Y 291.652,Z 250.655,A -85,B 0,C 180,E1 -16551.697,E2 -16551.697} C_VEL
LIN {X 0,Y 291.605,Z 250.658,A -85,B 0,C 180,E1 -16554.477,E2 -16554.477} C_VEL
LIN {X 0,Y 291.878,Z 250.624,A -85,B 0,C 180,E1 -16558.629,E2 -16558.629} C_VEL
LIN {X 0,Y 291.886,Z 250.62,A -85,B 0,C 180,E1 -16561.389,E2 -16561.389} C_VEL
LIN {X 0,Y 291.699,Z 250.639,A -85,B 0,C 180,E1 -16566.928,E2 -16566.928} C_VEL
LIN {X 0,Y 291.583,Z 250.659,A -85,B 0,C 180,E1 -16569.722,E2 -16569.722} C_VEL
LIN {X 0,Y 291.532,Z 250.668,A -85,B 0,C 180,E1 -16573.958,E2 -16573.958} C_VEL
LIN {X 0,Y 291.447,Z 250.674,A -85,B 0,C 180,E1 -16576.829,E2 -16576.829} C_VEL
LIN {X 0,Y 291.412,Z 250.675,A -85,B 0,C 180,E1 -16579.849,E2 -16579.849} C_VEL
LIN {X 0,Y 291.381,Z 250.687,A -85,B 0,C 180,E1 -16584.215,E2 -16584.215} C_VEL
LIN {X 0,Y 291.374,Z 250.685,A -85,B 0,C 180,E1 -16587.285,E2 -16587.285} C_VEL
LIN {X 0,Y 291.328,Z 250.69,A -85,B 0,C 180,E1 -16590.446,E2 -16590.446} C_VEL
LIN {X 0,Y 291.369,Z 250.689,A -85,B 0,C 180,E1 -16593.703,E2 -16593.703} C_VEL
LIN {X 0,Y 291.374,Z 250.687,A -85,B 0,C 180,E1 -16597.251,E2 -16597.251} C_VEL
LIN {X 0,Y 291.32,Z 250.694,A -85,B 0,C 180,E1 -16600.653,E2 -16600.653} C_VEL
LIN {X 0,Y 291.301,Z 250.697,A -85,B 0,C 180,E1 -16604.409,E2 -16604.409} C_VEL
LIN {X 0,Y 291.299,Z 250.698,A -85,B 0,C 180,E1 -16608.42,E2 -16608.42} C_VEL
LIN {X 0,Y 291.339,Z 250.693,A -85,B 0,C 180,E1 -16611.154,E2 -16611.154} C_VEL
LIN {X 0,Y 291.382,Z 250.689,A -85,B 0,C 180,E1 -16614.627,E2 -16614.627} C_VEL
LIN {X 0,Y 291.408,Z 250.8,A -85,B 0,C 180,E1 -16618.156,E2 -16618.156} C_VEL
LIN {X 0,Y 293.292,Z 259.99,A -85,B 0,C 180,E1 -16621.361,E2 -16621.361} C_VEL
LIN {X 0,Y 294.954,Z 268.282,A -85,B 0,C 180,E1 -16624.011,E2 -16624.011} C_VEL
LIN {X 0,Y 297.122,Z 275.756,A -85,B 0,C 180,E1 -16624.422,E2 -16624.422} C_VEL
LIN {X 0,Y 301.943,Z 307.858,A -85,B 0,C 180,E1 -16625.681,E2 -16625.681} C_VEL
LIN {X 0,Y 299.916,Z 375.86,A -85,B 0,C 180,E1 -16627.479,E2 -16627.479} C_VEL
LIN {X 0,Y 299.083,Z 389.407,A -85,B 0,C 180,E1 -16628.095,E2 -16628.095} C_VEL
LIN {X 0,Y 298.054,Z 401.835,A -85,B 0,C 180,E1 -16628.923,E2 -16628.923} C_VEL
LIN {X 0,Y 296.93,Z 413.038,A -85,B 0,C 180,E1 -16629.926,E2 -16629.926} C_VEL
LIN {X 0,Y 295.444,Z 424.691,A -85,B 0,C 180,E1 -16631.266,E2 -16631.266} C_VEL
LIN {X 0,Y 294.154,Z 435.825,A -85,B 0,C 180,E1 -16632.897,E2 -16632.897} C_VEL
LIN {X 0,Y 292.824,Z 445.54,A -85,B 0,C 180,E1 -16634.69,E2 -16634.69} C_VEL
LIN {X 0,Y 291.612,Z 454.555,A -85,B 0,C 180,E1 -16636.762,E2 -16636.762} C_VEL
LIN {X 0,Y 290.694,Z 461.757,A -85,B 0,C 180,E1 -16638.846,E2 -16638.846} C_VEL
LIN {X 0,Y 290.064,Z 467.482,A -85,B 0,C 180,E1 -16640.937,E2 -16640.937} C_VEL
LIN {X 0,Y 289.665,Z 471.962,A -85,B 0,C 180,E1 -16643.03,E2 -16643.03} C_VEL
LIN {X 0,Y 289.502,Z 474.453,A -85,B 0,C 180,E1 -16644.51,E2 -16644.51} C_VEL
LIN {X 0,Y 289.411,Z 476.233,A -85,B 0,C 180,E1 -16645.82,E2 -16645.82} C_VEL
LIN {X 0,Y 289.405,Z 477.664,A -85,B 0,C 180,E1 -16647.214,E2 -16647.214} C_VEL
LIN {X 0,Y 289.386,Z 478.672,A -85,B 0,C 180,E1 -16648.606,E2 -16648.606} C_VEL
LIN {X 0,Y 289.386,Z 479.278,A -85,B 0,C 180,E1 -16649.998,E2 -16649.998} C_VEL
LIN {X 0,Y 289.385,Z 479.479,A -85,B 0,C 180,E1 -16651.389,E2 -16651.389} C_VEL
LIN {X 0,Y 289.406,Z 479.233,A -85,B 0,C 180,E1 -16652.781,E2 -16652.781} C_VEL
LIN {X 0,Y 289.504,Z 477.554,A -85,B 0,C 180,E1 -16655.57,E2 -16655.57} C_VEL
LIN {X 0,Y 289.732,Z 476.108,A -85,B 0,C 180,E1 -16656.964,E2 -16656.964} C_VEL
LIN {X 0,Y 290.217,Z 473.102,A -85,B 0,C 180,E1 -16659.054,E2 -16659.054} C_VEL
LIN {X 0,Y 290.977,Z 469.051,A -85,B 0,C 180,E1 -16661.138,E2 -16661.138} C_VEL
LIN {X 0,Y 292.217,Z 462.841,A -85,B 0,C 180,E1 -16663.559,E2 -16663.559} C_VEL
LIN {X 0,Y 293.846,Z 456.077,A -85,B 0,C 180,E1 -16665.606,E2 -16665.606} C_VEL
LIN {X 0,Y 295.638,Z 447.717,A -85,B 0,C 180,E1 -16667.641,E2 -16667.641} C_VEL
LIN {X 0,Y 297.267,Z 439.154,A -85,B 0,C 180,E1 -16669.326,E2 -16669.326} C_VEL
LIN {X 0,Y 299.344,Z 428.662,A -85,B 0,C 180,E1 -16670.977,E2 -16670.977} C_VEL
LIN {X 0,Y 301.44,Z 416.918,A -85,B 0,C 180,E1 -16672.441,E2 -16672.441} C_VEL
LIN {X 0,Y 303.208,Z 405.187,A -85,B 0,C 180,E1 -16673.565,E2 -16673.565} C_VEL
LIN {X 0,Y 304.814,Z 391.957,A -85,B 0,C 180,E1 -16674.518,E2 -16674.518} C_VEL
LIN {X 0,Y 306.013,Z 379.357,A -85,B 0,C 180,E1 -16675.14,E2 -16675.14} C_VEL
LIN {X 0,Y 306.962,Z 360.932,A -85,B 0,C 180,E1 -16675.692,E2 -16675.692} C_VEL
LIN {X 0,Y 308.946,Z 309.844,A -85,B 0,C 180,E1 -16677.06,E2 -16677.06} C_VEL
LIN {X 0,Y 306.542,Z 294.799,A -85,B 0,C 180,E1 -16677.84,E2 -16677.84} C_VEL
LIN {X 0,Y 304.883,Z 287.013,A -85,B 0,C 180,E1 -16678.313,E2 -16678.313} C_VEL
LIN {X 0,Y 299.727,Z 275.182,A -85,B 0,C 180,E1 -16679.411,E2 -16679.411} C_VEL
LIN {X 0,Y 295.551,Z 266.75,A -85,B 0,C 180,E1 -16680.346,E2 -16680.346} C_VEL
LIN {X 0,Y 293.56,Z 258.58,A -85,B 0,C 180,E1 -16683.407,E2 -16683.407} C_VEL
LIN {X 0,Y 291.413,Z 250.872,A -85,B 0,C 180,E1 -16686.644,E2 -16686.644} C_VEL
LIN {X 0,Y 291.311,Z 250.697,A -85,B 0,C 180,E1 -16690.642,E2 -16690.642} C_VEL
LIN {X 0,Y 291.293,Z 250.702,A -85,B 0,C 180,E1 -16694.397,E2 -16694.397} C_VEL
LIN {X 0,Y 291.302,Z 250.696,A -85,B 0,C 180,E1 -16698.405,E2 -16698.405} C_VEL
LIN {X 0,Y 291.339,Z 250.69,A -85,B 0,C 180,E1 -16701.148,E2 -16701.148} C_VEL
LIN {X 0,Y 291.36,Z 250.69,A -85,B 0,C 180,E1 -16704.618,E2 -16704.618} C_VEL
LIN {X 0,Y 291.37,Z 250.688,A -85,B 0,C 180,E1 -16707.942,E2 -16707.942} C_VEL
LIN {X 0,Y 291.325,Z 250.693,A -85,B 0,C 180,E1 -16711.144,E2 -16711.144} C_VEL
LIN {X 0,Y 291.358,Z 250.684,A -85,B 0,C 180,E1 -16714.258,E2 -16714.258} C_VEL
LIN {X 0,Y 291.361,Z 250.683,A -85,B 0,C 180,E1 -16717.29,E2 -16717.29} C_VEL
LIN {X 0,Y 291.382,Z 250.683,A -85,B 0,C 180,E1 -16720.257,E2 -16720.257} C_VEL
LIN {X 0,Y 291.469,Z 250.67,A -85,B 0,C 180,E1 -16724.674,E2 -16724.674} C_VEL
LIN {X 0,Y 291.519,Z 250.668,A -85,B 0,C 180,E1 -16728.871,E2 -16728.871} C_VEL
LIN {X 0,Y 291.644,Z 250.651,A -85,B 0,C 180,E1 -16731.678,E2 -16731.678} C_VEL
LIN {X 0,Y 291.591,Z 250.656,A -85,B 0,C 180,E1 -16734.459,E2 -16734.459} C_VEL
LIN {X 0,Y 291.868,Z 250.629,A -85,B 0,C 180,E1 -16738.611,E2 -16738.611} C_VEL
LIN {X 0,Y 291.869,Z 250.631,A -85,B 0,C 180,E1 -16741.371,E2 -16741.371} C_VEL
LIN {X 0,Y 291.714,Z 250.646,A -85,B 0,C 180,E1 -16746.909,E2 -16746.909} C_VEL
LIN {X 0,Y 291.606,Z 250.664,A -85,B 0,C 180,E1 -16749.703,E2 -16749.703} C_VEL
LIN {X 0,Y 291.52,Z 250.814,A -85,B 0,C 180,E1 -16751.638,E2 -16751.638} C_VEL
LIN {X 0,Y 293.971,Z 259.653,A -85,B 0,C 180,E1 -16755.236,E2 -16755.236} C_VEL
LIN {X 0,Y 294.281,Z 260.685,A -85,B 0,C 180,E1 -16755.53,E2 -16755.53} C_VEL
LIN {X 0,Y 301.17,Z 273.959,A -85,B 0,C 180,E1 -16757.009,E2 -16757.009} C_VEL
LIN {X 0,Y 307.111,Z 287.27,A -85,B 0,C 180,E1 -16758.247,E2 -16758.247} C_VEL
LIN {X 0,Y 308.076,Z 290.761,A -85,B 0,C 180,E1 -16758.485,E2 -16758.485} C_VEL
LIN {X 0,Y 309.339,Z 298.25,A -85,B 0,C 180,E1 -16758.88,E2 -16758.88} C_VEL
LIN {X 0,Y 306.356,Z 369.149,A -85,B 0,C 180,E1 -16760.797,E2 -16760.797} C_VEL
LIN {X 0,Y 305.207,Z 383.002,A -85,B 0,C 180,E1 -16761.436,E2 -16761.436} C_VEL
LIN {X 0,Y 303.85,Z 395.679,A -85,B 0,C 180,E1 -16762.311,E2 -16762.311} C_VEL
LIN {X 0,Y 302.154,Z 407.903,A -85,B 0,C 180,E1 -16763.447,E2 -16763.447} C_VEL
LIN {X 0,Y 300.297,Z 418.854,A -85,B 0,C 180,E1 -16764.748,E2 -16764.748} C_VEL
LIN {X 0,Y 298.61,Z 427.956,A -85,B 0,C 180,E1 -16766.096,E2 -16766.096} C_VEL
LIN {X 0,Y 296.569,Z 437.766,A -85,B 0,C 180,E1 -16767.894,E2 -16767.894} C_VEL
LIN {X 0,Y 294.923,Z 445.473,A -85,B 0,C 180,E1 -16769.639,E2 -16769.639} C_VEL
LIN {X 0,Y 293.119,Z 453.255,A -85,B 0,C 180,E1 -16771.823,E2 -16771.823} C_VEL
LIN {X 0,Y 291.672,Z 459.868,A -85,B 0,C 180,E1 -16774.249,E2 -16774.249} C_VEL
LIN {X 0,Y 290.798,Z 463.988,A -85,B 0,C 180,E1 -16776.205,E2 -16776.205} C_VEL
LIN {X 0,Y 290.103,Z 467.129,A -85,B 0,C 180,E1 -16778.138,E2 -16778.138} C_VEL
LIN {X 0,Y 289.835,Z 468.376,A -85,B 0,C 180,E1 -16779.114,E2 -16779.114} C_VEL
LIN {X 0,Y 289.431,Z 470.304,A -85,B 0,C 180,E1 -16781.176,E2 -16781.176} C_VEL
LIN {X 0,Y 289.192,Z 471.315,A -85,B 0,C 180,E1 -16783.196,E2 -16783.196} C_VEL
LIN {X 0,Y 289.078,Z 471.488,A -85,B 0,C 180,E1 -16785.171,E2 -16785.171} C_VEL
LIN {X 0,Y 289.039,Z 470.883,A -85,B 0,C 180,E1 -16787.096,E2 -16787.096} C_VEL
LIN {X 0,Y 289.106,Z 469.522,A -85,B 0,C 180,E1 -16788.981,E2 -16788.981} C_VEL
LIN {X 0,Y 289.362,Z 467.196,A -85,B 0,C 180,E1 -16790.987,E2 -16790.987} C_VEL
LIN {X 0,Y 289.75,Z 463.649,A -85,B 0,C 180,E1 -16793.15,E2 -16793.15} C_VEL
LIN {X 0,Y 290.329,Z 458.77,A -85,B 0,C 180,E1 -16795.368,E2 -16795.368} C_VEL
LIN {X 0,Y 291.103,Z 452.212,A -85,B 0,C 180,E1 -16797.648,E2 -16797.648} C_VEL
LIN {X 0,Y 292.043,Z 444.968,A -85,B 0,C 180,E1 -16799.648,E2 -16799.648} C_VEL
LIN {X 0,Y 293.24,Z 436.208,A -85,B 0,C 180,E1 -16801.599,E2 -16801.599} C_VEL
LIN {X 0,Y 294.421,Z 427.184,A -85,B 0,C 180,E1 -16803.223,E2 -16803.223} C_VEL
LIN {X 0,Y 295.735,Z 417.21,A -85,B 0,C 180,E1 -16804.677,E2 -16804.677} C_VEL
LIN {X 0,Y 297.123,Z 404.907,A -85,B 0,C 180,E1 -16806.108,E2 -16806.108} C_VEL
LIN {X 0,Y 298.316,Z 392.515,A -85,B 0,C 180,E1 -16807.199,E2 -16807.199} C_VEL
LIN {X 0,Y 299.304,Z 379.198,A -85,B 0,C 180,E1 -16808.057,E2 -16808.057} C_VEL
LIN {X 0,Y 300.006,Z 366.608,A -85,B 0,C 180,E1 -16808.596,E2 -16808.596} C_VEL
LIN {X 0,Y 302.033,Z 294.341,A -85,B 0,C 180,E1 -16810.508,E2 -16810.508} C_VEL
LIN {X 0,Y 298.641,Z 275.777,A -85,B 0,C 180,E1 -16811.279,E2 -16811.279} C_VEL
LIN {X 0,Y 293.438,Z 260.872,A -85,B 0,C 180,E1 -16812.132,E2 -16812.132} C_VEL
LIN {X 0,Y 293.084,Z 259.254,A -85,B 0,C 180,E1 -16812.561,E2 -16812.561} C_VEL
LIN {X 0,Y 291.499,Z 250.731,A -85,B 0,C 180,E1 -16815.696,E2 -16815.696} C_VEL
LIN {X 0,Y 291.634,Z 250.658,A -85,B 0,C 180,E1 -16821.047,E2 -16821.047} C_VEL
LIN {X 0,Y 291.672,Z 250.654,A -85,B 0,C 180,E1 -16823.083,E2 -16823.083} C_VEL
LIN {X 0,Y 291.739,Z 250.645,A -85,B 0,C 180,E1 -16827.241,E2 -16827.241} C_VEL
LIN {X 0,Y 291.898,Z 250.62,A -85,B 0,C 180,E1 -16830.002,E2 -16830.002} C_VEL
LIN {X 0,Y 291.74,Z 250.645,A -85,B 0,C 180,E1 -16832.764,E2 -16832.764} C_VEL
LIN {X 0,Y 291.674,Z 250.652,A -85,B 0,C 180,E1 -16836.922,E2 -16836.922} C_VEL
LIN {X 0,Y 291.566,Z 250.66,A -85,B 0,C 180,E1 -16839.716,E2 -16839.716} C_VEL
LIN {X 0,Y 291.456,Z 250.679,A -85,B 0,C 180,E1 -16843.956,E2 -16843.956} C_VEL
LIN {X 0,Y 291.405,Z 250.677,A -85,B 0,C 180,E1 -16848.274,E2 -16848.274} C_VEL
LIN {X 0,Y 291.306,Z 250.695,A -85,B 0,C 180,E1 -16851.218,E2 -16851.218} C_VEL
LIN {X 0,Y 291.327,Z 250.694,A -85,B 0,C 180,E1 -16854.214,E2 -16854.214} C_VEL
LIN {X 0,Y 291.368,Z 250.683,A -85,B 0,C 180,E1 -16857.279,E2 -16857.279} C_VEL
LIN {X 0,Y 291.288,Z 250.695,A -85,B 0,C 180,E1 -16860.445,E2 -16860.445} C_VEL
LIN {X 0,Y 291.297,Z 250.697,A -85,B 0,C 180,E1 -16863.707,E2 -16863.707} C_VEL
LIN {X 0,Y 291.343,Z 250.69,A -85,B 0,C 180,E1 -16867.266,E2 -16867.266} C_VEL
LIN {X 0,Y 291.36,Z 250.692,A -85,B 0,C 180,E1 -16870.64,E2 -16870.64} C_VEL
LIN {X 0,Y 291.369,Z 250.692,A -85,B 0,C 180,E1 -16874.389,E2 -16874.389} C_VEL
LIN {X 0,Y 291.355,Z 250.69,A -85,B 0,C 180,E1 -16878.401,E2 -16878.401} C_VEL
LIN {X 0,Y 291.355,Z 250.691,A -85,B 0,C 180,E1 -16881.173,E2 -16881.173} C_VEL
LIN {X 0,Y 291.359,Z 250.69,A -85,B 0,C 180,E1 -16884.64,E2 -16884.64} C_VEL
LIN {X 0,Y 291.346,Z 250.69,A -85,B 0,C 180,E1 -16887.961,E2 -16887.961} C_VEL
LIN {X 0,Y 291.353,Z 250.693,A -85,B 0,C 180,E1 -16891.168,E2 -16891.168} C_VEL
LIN {X 0,Y 291.378,Z 250.686,A -85,B 0,C 180,E1 -16892.532,E2 -16892.532} C_VEL
LIN {X 0,Y 290.775,Z 250.766,A -85,B 0,C 180,E1 -16893.686,E2 -16893.686} C_VEL
LIN {X 0,Y 287.918,Z 251.123,A -85,B 0,C 180,E1 -16895.565,E2 -16895.565} C_VEL
LIN {X 0,Y 285.446,Z 251.428,A -85,B 0,C 180,E1 -16897.091,E2 -16897.091} C_VEL
LIN {X 0,Y 284.373,Z 251.559,A -85,B 0,C 180,E1 -16898.274,E2 -16898.274} C_VEL
LIN {X 0,Y 284.283,Z 251.568,A -85,B 0,C 180,E1 -16898.675,E2 -16898.675} C_VEL
LIN {X 0,Y 284.361,Z 251.558,A -85,B 0,C 180,E1 -16902.759,E2 -16902.759} C_VEL
LIN {X 0,Y 284.458,Z 251.551,A -85,B 0,C 180,E1 -16905.707,E2 -16905.707} C_VEL
LIN {X 0,Y 284.517,Z 251.542,A -85,B 0,C 180,E1 -16910.053,E2 -16910.053} C_VEL
LIN {X 0,Y 284.644,Z 251.52,A -85,B 0,C 180,E1 -16912.918,E2 -16912.918} C_VEL
LIN {X 0,Y 284.845,Z 251.501,A -85,B 0,C 180,E1 -16918.596,E2 -16918.596} C_VEL
LIN {X 0,Y 284.852,Z 251.496,A -85,B 0,C 180,E1 -16921.423,E2 -16921.423} C_VEL
LIN {X 0,Y 284.654,Z 251.515,A -85,B 0,C 180,E1 -16927.1,E2 -16927.1} C_VEL
LIN {X 0,Y 284.529,Z 251.538,A -85,B 0,C 180,E1 -16929.965,E2 -16929.965} C_VEL
LIN {X 0,Y 284.481,Z 251.549,A -85,B 0,C 180,E1 -16934.311,E2 -16934.311} C_VEL
LIN {X 0,Y 284.352,Z 251.555,A -85,B 0,C 180,E1 -16938.75,E2 -16938.75} C_VEL
LIN {X 0,Y 284.349,Z 251.564,A -85,B 0,C 180,E1 -16943.303,E2 -16943.303} C_VEL
LIN {X 0,Y 284.351,Z 251.56,A -85,B 0,C 180,E1 -16947.152,E2 -16947.152} C_VEL
LIN {X 0,Y 284.303,Z 251.572,A -85,B 0,C 180,E1 -16951.282,E2 -16951.282} C_VEL
LIN {X 0,Y 284.362,Z 251.559,A -85,B 0,C 180,E1 -16955.351,E2 -16955.351} C_VEL
LIN {X 0,Y 284.319,Z 251.566,A -85,B 0,C 180,E1 -16958.176,E2 -16958.176} C_VEL
LIN {X 0,Y 284.242,Z 251.573,A -85,B 0,C 180,E1 -16962.115,E2 -16962.115} C_VEL
LIN {X 0,Y 284.247,Z 251.574,A -85,B 0,C 180,E1 -16966.185,E2 -16966.185} C_VEL
LIN {X 0,Y 284.283,Z 251.574,A -85,B 0,C 180,E1 -16970.039,E2 -16970.039} C_VEL
LIN {X 0,Y 284.344,Z 251.568,A -85,B 0,C 180,E1 -16973.613,E2 -16973.613} C_VEL
LIN {X 0,Y 284.359,Z 251.631,A -85,B 0,C 180,E1 -16977.724,E2 -16977.724} C_VEL
LIN {X 0,Y 286.223,Z 260.572,A -85,B 0,C 180,E1 -16980.958,E2 -16980.958} C_VEL
LIN {X 0,Y 287.723,Z 268.065,A -85,B 0,C 180,E1 -16983.431,E2 -16983.431} C_VEL
LIN {X 0,Y 290.305,Z 275.963,A -85,B 0,C 180,E1 -16983.919,E2 -16983.919} C_VEL
LIN {X 0,Y 295.162,Z 307.877,A -85,B 0,C 180,E1 -16985.213,E2 -16985.213} C_VEL
LIN {X 0,Y 293.159,Z 376.037,A -85,B 0,C 180,E1 -16987.07,E2 -16987.07} C_VEL
LIN {X 0,Y 292.292,Z 389.481,A -85,B 0,C 180,E1 -16987.698,E2 -16987.698} C_VEL
LIN {X 0,Y 291.191,Z 402.396,A -85,B 0,C 180,E1 -16988.587,E2 -16988.587} C_VEL
LIN {X 0,Y 289.816,Z 415.009,A -85,B 0,C 180,E1 -16989.782,E2 -16989.782} C_VEL
LIN {X 0,Y 288.397,Z 426.307,A -85,B 0,C 180,E1 -16991.16,E2 -16991.16} C_VEL
LIN {X 0,Y 287.176,Z 436.065,A -85,B 0,C 180,E1 -16992.656,E2 -16992.656} C_VEL
LIN {X 0,Y 285.96,Z 444.876,A -85,B 0,C 180,E1 -16994.313,E2 -16994.313} C_VEL
LIN {X 0,Y 284.67,Z 453.988,A -85,B 0,C 180,E1 -16996.433,E2 -16996.433} C_VEL
LIN {X 0,Y 283.666,Z 461.302,A -85,B 0,C 180,E1 -16998.566,E2 -16998.566} C_VEL
LIN {X 0,Y 283.011,Z 467.107,A -85,B 0,C 180,E1 -17000.709,E2 -17000.709} C_VEL
LIN {X 0,Y 282.602,Z 471.654,A -85,B 0,C 180,E1 -17002.855,E2 -17002.855} C_VEL
LIN {X 0,Y 282.419,Z 474.458,A -85,B 0,C 180,E1 -17004.559,E2 -17004.559} C_VEL
LIN {X 0,Y 282.316,Z 477.471,A -85,B 0,C 180,E1 -17007.144,E2 -17007.144} C_VEL
LIN {X 0,Y 282.311,Z 478.505,A -85,B 0,C 180,E1 -17008.571,E2 -17008.571} C_VEL
LIN {X 0,Y 282.309,Z 479.137,A -85,B 0,C 180,E1 -17009.998,E2 -17009.998} C_VEL
LIN {X 0,Y 282.31,Z 479.373,A -85,B 0,C 180,E1 -17011.424,E2 -17011.424} C_VEL
LIN {X 0,Y 282.316,Z 479.176,A -85,B 0,C 180,E1 -17012.851,E2 -17012.851} C_VEL
LIN {X 0,Y 282.434,Z 477.556,A -85,B 0,C 180,E1 -17015.71,E2 -17015.71} C_VEL
LIN {X 0,Y 282.681,Z 476.151,A -85,B 0,C 180,E1 -17017.138,E2 -17017.138} C_VEL
LIN {X 0,Y 283.182,Z 473.196,A -85,B 0,C 180,E1 -17019.281,E2 -17019.281} C_VEL
LIN {X 0,Y 283.989,Z 469.206,A -85,B 0,C 180,E1 -17021.416,E2 -17021.416} C_VEL
LIN {X 0,Y 285.326,Z 463.091,A -85,B 0,C 180,E1 -17023.893,E2 -17023.893} C_VEL
LIN {X 0,Y 287.29,Z 455.174,A -85,B 0,C 180,E1 -17026.337,E2 -17026.337} C_VEL
LIN {X 0,Y 288.893,Z 448.174,A -85,B 0,C 180,E1 -17028.067,E2 -17028.067} C_VEL
LIN {X 0,Y 290.627,Z 439.788,A -85,B 0,C 180,E1 -17029.786,E2 -17029.786} C_VEL
LIN {X 0,Y 292.781,Z 429.474,A -85,B 0,C 180,E1 -17031.47,E2 -17031.47} C_VEL
LIN {X 0,Y 294.744,Z 419.33,A -85,B 0,C 180,E1 -17032.794,E2 -17032.794} C_VEL
LIN {X 0,Y 296.492,Z 408.358,A -85,B 0,C 180,E1 -17033.946,E2 -17033.946} C_VEL
LIN {X 0,Y 298.173,Z 396.282,A -85,B 0,C 180,E1 -17034.915,E2 -17034.915} C_VEL
LIN {X 0,Y 299.581,Z 382.976,A -85,B 0,C 180,E1 -17035.672,E2 -17035.672} C_VEL
LIN {X 0,Y 300.533,Z 370.104,A -85,B 0,C 180,E1 -17036.143,E2 -17036.143} C_VEL
LIN {X 0,Y 302.958,Z 310.303,A -85,B 0,C 180,E1 -17037.791,E2 -17037.791} C_VEL
LIN {X 0,Y 300.062,Z 292.696,A -85,B 0,C 180,E1 -17038.767,E2 -17038.767} C_VEL
LIN {X 0,Y 298.825,Z 288.576,A -85,B 0,C 180,E1 -17039.077,E2 -17039.077} C_VEL
LIN {X 0,Y 293.889,Z 277.661,A -85,B 0,C 180,E1 -17040.169,E2 -17040.169} C_VEL
LIN {X 0,Y 289.594,Z 269.289,A -85,B 0,C 180,E1 -17041.154,E2 -17041.154} C_VEL
LIN {X 0,Y 288.291,Z 266.379,A -85,B 0,C 180,E1 -17041.524,E2 -17041.524} C_VEL
LIN {X 0,Y 286.175,Z 258.178,A -85,B 0,C 180,E1 -17044.823,E2 -17044.823} C_VEL
LIN {X 0,Y 284.301,Z 251.651,A -85,B 0,C 180,E1 -17047.803,E2 -17047.803} C_VEL
LIN {X 0,Y 284.295,Z 251.573,A -85,B 0,C 180,E1 -17049.993,E2 -17049.993} C_VEL
LIN {X 0,Y 284.244,Z 251.579,A -85,B 0,C 180,E1 -17054.181,E2 -17054.181} C_VEL
LIN {X 0,Y 284.247,Z 251.574,A -85,B 0,C 180,E1 -17058.111,E2 -17058.111} C_VEL
LIN {X 0,Y 284.301,Z 251.571,A -85,B 0,C 180,E1 -17061.821,E2 -17061.821} C_VEL
LIN {X 0,Y 284.313,Z 251.57,A -85,B 0,C 180,E1 -17065.343,E2 -17065.343} C_VEL
LIN {X 0,Y 284.283,Z 251.574,A -85,B 0,C 180,E1 -17068.716,E2 -17068.716} C_VEL
LIN {X 0,Y 284.329,Z 251.562,A -85,B 0,C 180,E1 -17072.846,E2 -17072.846} C_VEL
LIN {X 0,Y 284.327,Z 251.561,A -85,B 0,C 180,E1 -17076.695,E2 -17076.695} C_VEL
LIN {X 0,Y 284.332,Z 251.564,A -85,B 0,C 180,E1 -17079.92,E2 -17079.92} C_VEL
LIN {X 0,Y 284.41,Z 251.549,A -85,B 0,C 180,E1 -17084.508,E2 -17084.508} C_VEL
LIN {X 0,Y 284.451,Z 251.546,A -85,B 0,C 180,E1 -17088.591,E2 -17088.591} C_VEL
LIN {X 0,Y 284.601,Z 251.527,A -85,B 0,C 180,E1 -17091.471,E2 -17091.471} C_VEL
LIN {X 0,Y 284.561,Z 251.532,A -85,B 0,C 180,E1 -17094.322,E2 -17094.322} C_VEL
LIN {X 0,Y 284.833,Z 251.505,A -85,B 0,C 180,E1 -17098.577,E2 -17098.577} C_VEL
LIN {X 0,Y 284.836,Z 251.506,A -85,B 0,C 180,E1 -17101.404,E2 -17101.404} C_VEL
LIN {X 0,Y 284.667,Z 251.524,A -85,B 0,C 180,E1 -17107.081,E2 -17107.081} C_VEL
LIN {X 0,Y 284.511,Z 251.6,A -85,B 0,C 180,E1 -17110.486,E2 -17110.486} C_VEL
LIN {X 0,Y 285.887,Z 256.631,A -85,B 0,C 180,E1 -17112.772,E2 -17112.772} C_VEL
LIN {X 0,Y 287.031,Z 260.591,A -85,B 0,C 180,E1 -17114.343,E2 -17114.343} C_VEL
LIN {X 0,Y 294.085,Z 273.831,A -85,B 0,C 180,E1 -17115.985,E2 -17115.985} C_VEL
LIN {X 0,Y 299.716,Z 285.752,A -85,B 0,C 180,E1 -17117.211,E2 -17117.211} C_VEL
LIN {X 0,Y 302.23,Z 292.244,A -85,B 0,C 180,E1 -17117.771,E2 -17117.771} C_VEL
LIN {X 0,Y 303.423,Z 299.251,A -85,B 0,C 180,E1 -17118.162,E2 -17118.162} C_VEL
LIN {X 0,Y 300.312,Z 369.097,A -85,B 0,C 180,E1 -17120.099,E2 -17120.099} C_VEL
LIN {X 0,Y 299.185,Z 382.305,A -85,B 0,C 180,E1 -17120.71,E2 -17120.71} C_VEL
LIN {X 0,Y 297.844,Z 394.444,A -85,B 0,C 180,E1 -17121.533,E2 -17121.533} C_VEL
LIN {X 0,Y 296.06,Z 407.011,A -85,B 0,C 180,E1 -17122.692,E2 -17122.692} C_VEL
LIN {X 0,Y 294.005,Z 418.67,A -85,B 0,C 180,E1 -17124.082,E2 -17124.082} C_VEL
LIN {X 0,Y 291.964,Z 429.062,A -85,B 0,C 180,E1 -17125.664,E2 -17125.664} C_VEL
LIN {X 0,Y 289.931,Z 438.269,A -85,B 0,C 180,E1 -17127.411,E2 -17127.411} C_VEL
LIN {X 0,Y 287.821,Z 447.485,A -85,B 0,C 180,E1 -17129.607,E2 -17129.607} C_VEL
LIN {X 0,Y 285.957,Z 454.923,A -85,B 0,C 180,E1 -17131.885,E2 -17131.885} C_VEL
LIN {X 0,Y 284.819,Z 459.905,A -85,B 0,C 180,E1 -17133.804,E2 -17133.804} C_VEL
LIN {X 0,Y 283.597,Z 465.224,A -85,B 0,C 180,E1 -17136.481,E2 -17136.481} C_VEL
LIN {X 0,Y 282.943,Z 467.933,A -85,B 0,C 180,E1 -17138.372,E2 -17138.372} C_VEL
LIN {X 0,Y 282.464,Z 469.915,A -85,B 0,C 180,E1 -17140.293,E2 -17140.293} C_VEL
LIN {X 0,Y 282.194,Z 471.165,A -85,B 0,C 180,E1 -17142.239,E2 -17142.239} C_VEL
LIN {X 0,Y 282.011,Z 471.627,A -85,B 0,C 180,E1 -17144.233,E2 -17144.233} C_VEL
LIN {X 0,Y 281.957,Z 471.289,A -85,B 0,C 180,E1 -17146.272,E2 -17146.272} C_VEL
LIN {X 0,Y 281.959,Z 470.073,A -85,B 0,C 180,E1 -17148.379,E2 -17148.379} C_VEL
LIN {X 0,Y 282.196,Z 467.903,A -85,B 0,C 180,E1 -17150.518,E2 -17150.518} C_VEL
LIN {X 0,Y 282.587,Z 464.629,A -85,B 0,C 180,E1 -17152.715,E2 -17152.715} C_VEL
LIN {X 0,Y 283.16,Z 459.545,A -85,B 0,C 180,E1 -17155.194,E2 -17155.194} C_VEL
LIN {X 0,Y 283.883,Z 453.915,A -85,B 0,C 180,E1 -17157.299,E2 -17157.299} C_VEL
LIN {X 0,Y 284.711,Z 447.403,A -85,B 0,C 180,E1 -17159.258,E2 -17159.258} C_VEL
LIN {X 0,Y 285.939,Z 438.864,A -85,B 0,C 180,E1 -17161.319,E2 -17161.319} C_VEL
LIN {X 0,Y 287.301,Z 428.647,A -85,B 0,C 180,E1 -17163.292,E2 -17163.292} C_VEL
LIN {X 0,Y 288.653,Z 419.001,A -85,B 0,C 180,E1 -17164.784,E2 -17164.784} C_VEL
LIN {X 0,Y 289.88,Z 408.569,A -85,B 0,C 180,E1 -17166.088,E2 -17166.088} C_VEL
LIN {X 0,Y 291.18,Z 396.321,A -85,B 0,C 180,E1 -17167.286,E2 -17167.286} C_VEL
LIN {X 0,Y 292.186,Z 383.863,A -85,B 0,C 180,E1 -17168.206,E2 -17168.206} C_VEL
LIN {X 0,Y 293.04,Z 370.055,A -85,B 0,C 180,E1 -17168.895,E2 -17168.895} C_VEL
LIN {X 0,Y 293.88,Z 346.953,A -85,B 0,C 180,E1 -17169.563,E2 -17169.563} C_VEL
LIN {X 0,Y 295.289,Z 294.844,A -85,B 0,C 180,E1 -17170.969,E2 -17170.969} C_VEL
LIN {X 0,Y 292.261,Z 278.195,A -85,B 0,C 180,E1 -17171.675,E2 -17171.675} C_VEL
LIN {X 0,Y 286.19,Z 260.849,A -85,B 0,C 180,E1 -17172.699,E2 -17172.699} C_VEL
LIN {X 0,Y 285.326,Z 256.194,A -85,B 0,C 180,E1 -17174.282,E2 -17174.282} C_VEL
LIN {X 0,Y 284.441,Z 251.612,A -85,B 0,C 180,E1 -17176.063,E2 -17176.063} C_VEL
LIN {X 0,Y 284.596,Z 251.536,A -85,B 0,C 180,E1 -17180.951,E2 -17180.951} C_VEL
LIN {X 0,Y 284.535,Z 251.542,A -85,B 0,C 180,E1 -17184.332,E2 -17184.332} C_VEL
LIN {X 0,Y 284.794,Z 251.51,A -85,B 0,C 180,E1 -17188.588,E2 -17188.588} C_VEL
LIN {X 0,Y 284.794,Z 251.51,A -85,B 0,C 180,E1 -17191.416,E2 -17191.416} C_VEL
LIN {X 0,Y 284.537,Z 251.54,A -85,B 0,C 180,E1 -17195.672,E2 -17195.672} C_VEL
LIN {X 0,Y 284.599,Z 251.534,A -85,B 0,C 180,E1 -17199.052,E2 -17199.052} C_VEL
LIN {X 0,Y 284.412,Z 251.554,A -85,B 0,C 180,E1 -17202.852,E2 -17202.852} C_VEL
LIN {X 0,Y 284.392,Z 251.557,A -85,B 0,C 180,E1 -17205.776,E2 -17205.776} C_VEL
LIN {X 0,Y 284.32,Z 251.565,A -85,B 0,C 180,E1 -17210.249,E2 -17210.249} C_VEL
LIN {X 0,Y 284.283,Z 251.569,A -85,B 0,C 180,E1 -17214.854,E2 -17214.854} C_VEL
LIN {X 0,Y 284.278,Z 251.562,A -85,B 0,C 180,E1 -17218.019,E2 -17218.019} C_VEL
LIN {X 0,Y 284.247,Z 251.57,A -85,B 0,C 180,E1 -17221.282,E2 -17221.282} C_VEL
LIN {X 0,Y 284.315,Z 251.567,A -85,B 0,C 180,E1 -17225.362,E2 -17225.362} C_VEL
LIN {X 0,Y 284.284,Z 251.572,A -85,B 0,C 180,E1 -17228.176,E2 -17228.176} C_VEL
LIN {X 0,Y 284.303,Z 251.57,A -85,B 0,C 180,E1 -17232.15,E2 -17232.15} C_VEL
LIN {X 0,Y 284.317,Z 251.566,A -85,B 0,C 180,E1 -17236.218,E2 -17236.218} C_VEL
LIN {X 0,Y 284.321,Z 251.566,A -85,B 0,C 180,E1 -17240.023,E2 -17240.023} C_VEL
LIN {X 0,Y 284.328,Z 251.562,A -85,B 0,C 180,E1 -17243.628,E2 -17243.628} C_VEL
LIN {X 0,Y 284.283,Z 251.573,A -85,B 0,C 180,E1 -17247.201,E2 -17247.201} C_VEL
LIN {X 0,Y 284.334,Z 251.565,A -85,B 0,C 180,E1 -17250.386,E2 -17250.386} C_VEL
LIN {X 0,Y 284.356,Z 251.558,A -85,B 0,C 180,E1 -17253.597,E2 -17253.597} C_VEL
LIN {X 0,Y 284.318,Z 251.565,A -85,B 0,C 180,E1 -17256.715,E2 -17256.715} C_VEL
LIN {X 0,Y 284.283,Z 251.568,A -85,B 0,C 180,E1 -17258.675,E2 -17258.675} C_VEL
LIN {X 0,Y 283.615,Z 251.656,A -85,B 0,C 180,E1 -17259.857,E2 -17259.857} C_VEL
LIN {X 0,Y 280.802,Z 252.003,A -85,B 0,C 180,E1 -17261.785,E2 -17261.785} C_VEL
LIN {X 0,Y 278.441,Z 252.298,A -85,B 0,C 180,E1 -17263.351,E2 -17263.351} C_VEL
LIN {X 0,Y 277.453,Z 252.416,A -85,B 0,C 180,E1 -17264.563,E2 -17264.563} C_VEL
LIN {X 0,Y 277.386,Z 252.425,A -85,B 0,C 180,E1 -17264.973,E2 -17264.973} C_VEL
LIN {X 0,Y 277.431,Z 252.424,A -85,B 0,C 180,E1 -17268.318,E2 -17268.318} C_VEL
LIN {X 0,Y 277.571,Z 252.406,A -85,B 0,C 180,E1 -17271.272,E2 -17271.272} C_VEL
LIN {X 0,Y 277.544,Z 252.411,A -85,B 0,C 180,E1 -17274.197,E2 -17274.197} C_VEL
LIN {X 0,Y 277.812,Z 252.377,A -85,B 0,C 180,E1 -17278.56,E2 -17278.56} C_VEL
LIN {X 0,Y 277.818,Z 252.372,A -85,B 0,C 180,E1 -17281.459,E2 -17281.459} C_VEL
LIN {X 0,Y 277.613,Z 252.391,A -85,B 0,C 180,E1 -17287.281,E2 -17287.281} C_VEL
LIN {X 0,Y 277.47,Z 252.419,A -85,B 0,C 180,E1 -17290.222,E2 -17290.222} C_VEL
LIN {X 0,Y 277.427,Z 252.426,A -85,B 0,C 180,E1 -17294.683,E2 -17294.683} C_VEL
LIN {X 0,Y 277.305,Z 252.432,A -85,B 0,C 180,E1 -17299.245,E2 -17299.245} C_VEL
LIN {X 0,Y 277.304,Z 252.44,A -85,B 0,C 180,E1 -17303.931,E2 -17303.931} C_VEL
LIN {X 0,Y 277.29,Z 252.437,A -85,B 0,C 180,E1 -17307.487,E2 -17307.487} C_VEL
LIN {X 0,Y 277.263,Z 252.445,A -85,B 0,C 180,E1 -17312.17,E2 -17312.17} C_VEL
LIN {X 0,Y 277.297,Z 252.435,A -85,B 0,C 180,E1 -17315.8,E2 -17315.8} C_VEL
LIN {X 0,Y 277.242,Z 252.452,A -85,B 0,C 180,E1 -17319.336,E2 -17319.336} C_VEL
LIN {X 0,Y 277.182,Z 252.454,A -85,B 0,C 180,E1 -17323.213,E2 -17323.213} C_VEL
LIN {X 0,Y 277.182,Z 252.454,A -85,B 0,C 180,E1 -17327.342,E2 -17327.342} C_VEL
LIN {X 0,Y 277.251,Z 252.451,A -85,B 0,C 180,E1 -17331.806,E2 -17331.806} C_VEL
LIN {X 0,Y 277.304,Z 252.445,A -85,B 0,C 180,E1 -17334.342,E2 -17334.342} C_VEL
LIN {X 0,Y 277.308,Z 252.576,A -85,B 0,C 180,E1 -17337.392,E2 -17337.392} C_VEL
LIN {X 0,Y 279.38,Z 262.548,A -85,B 0,C 180,E1 -17341.034,E2 -17341.034} C_VEL
LIN {X 0,Y 280.47,Z 268.055,A -85,B 0,C 180,E1 -17342.872,E2 -17342.872} C_VEL
LIN {X 0,Y 284.056,Z 279.02,A -85,B 0,C 180,E1 -17343.538,E2 -17343.538} C_VEL
LIN {X 0,Y 288.53,Z 309.602,A -85,B 0,C 180,E1 -17344.792,E2 -17344.792} C_VEL
LIN {X 0,Y 286.404,Z 375.918,A -85,B 0,C 180,E1 -17346.641,E2 -17346.641} C_VEL
LIN {X 0,Y 285.528,Z 389.35,A -85,B 0,C 180,E1 -17347.284,E2 -17347.284} C_VEL
LIN {X 0,Y 284.464,Z 401.735,A -85,B 0,C 180,E1 -17348.15,E2 -17348.15} C_VEL
LIN {X 0,Y 283.112,Z 413.689,A -85,B 0,C 180,E1 -17349.281,E2 -17349.281} C_VEL
LIN {X 0,Y 281.58,Z 425.193,A -85,B 0,C 180,E1 -17350.686,E2 -17350.686} C_VEL
LIN {X 0,Y 280.345,Z 434.959,A -85,B 0,C 180,E1 -17352.185,E2 -17352.185} C_VEL
LIN {X 0,Y 279.107,Z 444.145,A -85,B 0,C 180,E1 -17353.917,E2 -17353.917} C_VEL
LIN {X 0,Y 277.712,Z 453.36,A -85,B 0,C 180,E1 -17356.087,E2 -17356.087} C_VEL
LIN {X 0,Y 276.651,Z 460.776,A -85,B 0,C 180,E1 -17358.272,E2 -17358.272} C_VEL
LIN {X 0,Y 275.978,Z 466.692,A -85,B 0,C 180,E1 -17360.47,E2 -17360.47} C_VEL
LIN {X 0,Y 275.535,Z 471.315,A -85,B 0,C 180,E1 -17362.67,E2 -17362.67} C_VEL
LIN {X 0,Y 275.325,Z 474.473,A -85,B 0,C 180,E1 -17364.635,E2 -17364.635} C_VEL
LIN {X 0,Y 275.228,Z 477.257,A -85,B 0,C 180,E1 -17367.07,E2 -17367.07} C_VEL
LIN {X 0,Y 275.238,Z 478.328,A -85,B 0,C 180,E1 -17368.534,E2 -17368.534} C_VEL
LIN {X 0,Y 275.234,Z 478.992,A -85,B 0,C 180,E1 -17369.998,E2 -17369.998} C_VEL
LIN {X 0,Y 275.237,Z 479.258,A -85,B 0,C 180,E1 -17371.461,E2 -17371.461} C_VEL
LIN {X 0,Y 275.229,Z 479.117,A -85,B 0,C 180,E1 -17372.925,E2 -17372.925} C_VEL
LIN {X 0,Y 275.364,Z 477.559,A -85,B 0,C 180,E1 -17375.857,E2 -17375.857} C_VEL
LIN {X 0,Y 275.626,Z 476.183,A -85,B 0,C 180,E1 -17377.322,E2 -17377.322} C_VEL
LIN {X 0,Y 276.166,Z 473.287,A -85,B 0,C 180,E1 -17379.519,E2 -17379.519} C_VEL
LIN {X 0,Y 277.019,Z 469.371,A -85,B 0,C 180,E1 -17381.707,E2 -17381.707} C_VEL
LIN {X 0,Y 278.202,Z 464.336,A -85,B 0,C 180,E1 -17383.883,E2 -17383.883} C_VEL
LIN {X 0,Y 279.877,Z 458.024,A -85,B 0,C 180,E1 -17386.032,E2 -17386.032} C_VEL
LIN {X 0,Y 281.82,Z 450.319,A -85,B 0,C 180,E1 -17388.118,E2 -17388.118} C_VEL
LIN {X 0,Y 283.58,Z 442.346,A -85,B 0,C 180,E1 -17389.883,E2 -17389.883} C_VEL
LIN {X 0,Y 285.778,Z 432.458,A -85,B 0,C 180,E1 -17391.644,E2 -17391.644} C_VEL
LIN {X 0,Y 287.739,Z 423.002,A -85,B 0,C 180,E1 -17393.001,E2 -17393.001} C_VEL
LIN {X 0,Y 289.795,Z 411.387,A -85,B 0,C 180,E1 -17394.345,E2 -17394.345} C_VEL
LIN {X 0,Y 291.756,Z 399.114,A -85,B 0,C 180,E1 -17395.406,E2 -17395.406} C_VEL
LIN {X 0,Y 293.229,Z 386.518,A -85,B 0,C 180,E1 -17396.222,E2 -17396.222} C_VEL
LIN {X 0,Y 294.406,Z 373.363,A -85,B 0,C 180,E1 -17396.778,E2 -17396.778} C_VEL
LIN {X 0,Y 297.042,Z 311.165,A -85,B 0,C 180,E1 -17398.547,E2 -17398.547} C_VEL
LIN {X 0,Y 294.29,Z 294.311,A -85,B 0,C 180,E1 -17399.515,E2 -17399.515} C_VEL
LIN {X 0,Y 292.109,Z 288.612,A -85,B 0,C 180,E1 -17400.043,E2 -17400.043} C_VEL
LIN {X 0,Y 286.992,Z 277.707,A -85,B 0,C 180,E1 -17401.251,E2 -17401.251} C_VEL
LIN {X 0,Y 282.989,Z 270.14,A -85,B 0,C 180,E1 -17402.216,E2 -17402.216} C_VEL
LIN {X 0,Y 281.074,Z 266.224,A -85,B 0,C 180,E1 -17402.763,E2 -17402.763} C_VEL
LIN {X 0,Y 278.885,Z 258.103,A -85,B 0,C 180,E1 -17406.243,E2 -17406.243} C_VEL
LIN {X 0,Y 277.25,Z 252.497,A -85,B 0,C 180,E1 -17409.009,E2 -17409.009} C_VEL
LIN {X 0,Y 277.202,Z 252.452,A -85,B 0,C 180,E1 -17413.195,E2 -17413.195} C_VEL
LIN {X 0,Y 277.201,Z 252.454,A -85,B 0,C 180,E1 -17417.324,E2 -17417.324} C_VEL
LIN {X 0,Y 277.255,Z 252.448,A -85,B 0,C 180,E1 -17421.79,E2 -17421.79} C_VEL
LIN {X 0,Y 277.282,Z 252.44,A -85,B 0,C 180,E1 -17424.332,E2 -17424.332} C_VEL
LIN {X 0,Y 277.242,Z 252.448,A -85,B 0,C 180,E1 -17427.827,E2 -17427.827} C_VEL
LIN {X 0,Y 277.268,Z 252.445,A -85,B 0,C 180,E1 -17432.511,E2 -17432.511} C_VEL
LIN {X 0,Y 277.282,Z 252.444,A -85,B 0,C 180,E1 -17436.067,E2 -17436.067} C_VEL
LIN {X 0,Y 277.271,Z 252.438,A -85,B 0,C 180,E1 -17440.752,E2 -17440.752} C_VEL
LIN {X 0,Y 277.376,Z 252.429,A -85,B 0,C 180,E1 -17445.314,E2 -17445.314} C_VEL
LIN {X 0,Y 277.445,Z 252.425,A -85,B 0,C 180,E1 -17449.777,E2 -17449.777} C_VEL
LIN {X 0,Y 277.594,Z 252.407,A -85,B 0,C 180,E1 -17452.718,E2 -17452.718} C_VEL
LIN {X 0,Y 277.799,Z 252.382,A -85,B 0,C 180,E1 -17458.541,E2 -17458.541} C_VEL
LIN {X 0,Y 277.802,Z 252.382,A -85,B 0,C 180,E1 -17461.44,E2 -17461.44} C_VEL
LIN {X 0,Y 277.623,Z 252.402,A -85,B 0,C 180,E1 -17467.262,E2 -17467.262} C_VEL
LIN {X 0,Y 277.593,Z 252.627,A -85,B 0,C 180,E1 -17469.469,E2 -17469.469} C_VEL
LIN {X 0,Y 279.78,Z 260.61,A -85,B 0,C 180,E1 -17473.056,E2 -17473.056} C_VEL
LIN {X 0,Y 285.522,Z 270.942,A -85,B 0,C 180,E1 -17474.512,E2 -17474.512} C_VEL
LIN {X 0,Y 291.117,Z 281.871,A -85,B 0,C 180,E1 -17475.823,E2 -17475.823} C_VEL
LIN {X 0,Y 296.426,Z 294.114,A -85,B 0,C 180,E1 -17477.041,E2 -17477.041} C_VEL
LIN {X 0,Y 297.543,Z 300.911,A -85,B 0,C 180,E1 -17477.429,E2 -17477.429} C_VEL
LIN {X 0,Y 294.341,Z 369.293,A -85,B 0,C 180,E1 -17479.365,E2 -17479.365} C_VEL
LIN {X 0,Y 293.108,Z 383.026,A -85,B 0,C 180,E1 -17480.021,E2 -17480.021} C_VEL
LIN {X 0,Y 291.686,Z 394.948,A -85,B 0,C 180,E1 -17480.854,E2 -17480.854} C_VEL
LIN {X 0,Y 289.762,Z 407.705,A -85,B 0,C 180,E1 -17482.071,E2 -17482.071} C_VEL
LIN {X 0,Y 287.779,Z 418.348,A -85,B 0,C 180,E1 -17483.37,E2 -17483.37} C_VEL
LIN {X 0,Y 285.723,Z 428.393,A -85,B 0,C 180,E1 -17484.9,E2 -17484.9} C_VEL
LIN {X 0,Y 283.429,Z 438.283,A -85,B 0,C 180,E1 -17486.797,E2 -17486.797} C_VEL
LIN {X 0,Y 281.239,Z 447.401,A -85,B 0,C 180,E1 -17489.006,E2 -17489.006} C_VEL
LIN {X 0,Y 279.341,Z 454.517,A -85,B 0,C 180,E1 -17491.201,E2 -17491.201} C_VEL
LIN {X 0,Y 277.698,Z 461.048,A -85,B 0,C 180,E1 -17493.819,E2 -17493.819} C_VEL
LIN {X 0,Y 276.412,Z 466.202,A -85,B 0,C 180,E1 -17496.677,E2 -17496.677} C_VEL
LIN {X 0,Y 275.519,Z 469.692,A -85,B 0,C 180,E1 -17499.605,E2 -17499.605} C_VEL
LIN {X 0,Y 275.099,Z 471.335,A -85,B 0,C 180,E1 -17502.199,E2 -17502.199} C_VEL
LIN {X 0,Y 274.906,Z 471.75,A -85,B 0,C 180,E1 -17504.294,E2 -17504.294} C_VEL
LIN {X 0,Y 274.852,Z 471.321,A -85,B 0,C 180,E1 -17506.343,E2 -17506.343} C_VEL
LIN {X 0,Y 274.868,Z 470.145,A -85,B 0,C 180,E1 -17508.338,E2 -17508.338} C_VEL
LIN {X 0,Y 275.075,Z 468.239,A -85,B 0,C 180,E1 -17510.306,E2 -17510.306} C_VEL
LIN {X 0,Y 275.398,Z 465.536,A -85,B 0,C 180,E1 -17512.268,E2 -17512.268} C_VEL
LIN {X 0,Y 275.913,Z 461.251,A -85,B 0,C 180,E1 -17514.575,E2 -17514.575} C_VEL
LIN {X 0,Y 276.657,Z 455.448,A -85,B 0,C 180,E1 -17516.938,E2 -17516.938} C_VEL
LIN {X 0,Y 277.631,Z 447.801,A -85,B 0,C 180,E1 -17519.368,E2 -17519.368} C_VEL
LIN {X 0,Y 278.855,Z 439.75,A -85,B 0,C 180,E1 -17521.392,E2 -17521.392} C_VEL
LIN {X 0,Y 280.021,Z 431.173,A -85,B 0,C 180,E1 -17523.146,E2 -17523.146} C_VEL
LIN {X 0,Y 281.553,Z 420.569,A -85,B 0,C 180,E1 -17524.894,E2 -17524.894} C_VEL
LIN {X 0,Y 282.97,Z 409.135,A -85,B 0,C 180,E1 -17526.394,E2 -17526.394} C_VEL
LIN {X 0,Y 284.378,Z 396.415,A -85,B 0,C 180,E1 -17527.671,E2 -17527.671} C_VEL
LIN {X 0,Y 285.39,Z 384.027,A -85,B 0,C 180,E1 -17528.609,E2 -17528.609} C_VEL
LIN {X 0,Y 286.25,Z 371.252,A -85,B 0,C 180,E1 -17529.273,E2 -17529.273} C_VEL
LIN {X 0,Y 287.04,Z 351.554,A -85,B 0,C 180,E1 -17529.879,E2 -17529.879} C_VEL
LIN {X 0,Y 288.678,Z 296.108,A -85,B 0,C 180,E1 -17531.411,E2 -17531.411} C_VEL
LIN {X 0,Y 285.919,Z 280.695,A -85,B 0,C 180,E1 -17532.081,E2 -17532.081} C_VEL
LIN {X 0,Y 279.042,Z 260.977,A -85,B 0,C 180,E1 -17533.276,E2 -17533.276} C_VEL
LIN {X 0,Y 278.295,Z 257.035,A -85,B 0,C 180,E1 -17534.626,E2 -17534.626} C_VEL
LIN {X 0,Y 277.402,Z 252.478,A -85,B 0,C 180,E1 -17536.449,E2 -17536.449} C_VEL
LIN {X 0,Y 277.544,Z 252.412,A -85,B 0,C 180,E1 -17541.264,E2 -17541.264} C_VEL
LIN {X 0,Y 277.505,Z 252.417,A -85,B 0,C 180,E1 -17544.188,E2 -17544.188} C_VEL
LIN {X 0,Y 277.76,Z 252.386,A -85,B 0,C 180,E1 -17548.553,E2 -17548.553} C_VEL
LIN {X 0,Y 277.76,Z 252.386,A -85,B 0,C 180,E1 -17551.452,E2 -17551.452} C_VEL
LIN {X 0,Y 277.582,Z 252.41,A -85,B 0,C 180,E1 -17557.275,E2 -17557.275} C_VEL
LIN {X 0,Y 277.444,Z 252.416,A -85,B 0,C 180,E1 -17560.216,E2 -17560.216} C_VEL
LIN {X 0,Y 277.355,Z 252.434,A -85,B 0,C 180,E1 -17564.681,E2 -17564.681} C_VEL
LIN {X 0,Y 277.283,Z 252.436,A -85,B 0,C 180,E1 -17569.241,E2 -17569.241} C_VEL
LIN {X 0,Y 277.237,Z 252.45,A -85,B 0,C 180,E1 -17574.164,E2 -17574.164} C_VEL
LIN {X 0,Y 277.272,Z 252.439,A -85,B 0,C 180,E1 -17577.512,E2 -17577.512} C_VEL
LIN {X 0,Y 277.223,Z 252.445,A -85,B 0,C 180,E1 -17580.49,E2 -17580.49} C_VEL
LIN {X 0,Y 277.208,Z 252.454,A -85,B 0,C 180,E1 -17583.904,E2 -17583.904} C_VEL
LIN {X 0,Y 277.235,Z 252.447,A -85,B 0,C 180,E1 -17587.477,E2 -17587.477} C_VEL
LIN {X 0,Y 277.225,Z 252.449,A -85,B 0,C 180,E1 -17591.236,E2 -17591.236} C_VEL
LIN {X 0,Y 277.251,Z 252.444,A -85,B 0,C 180,E1 -17595.219,E2 -17595.219} C_VEL
LIN {X 0,Y 277.264,Z 252.444,A -85,B 0,C 180,E1 -17599.505,E2 -17599.505} C_VEL
LIN {X 0,Y 277.262,Z 252.448,A -85,B 0,C 180,E1 -17602.545,E2 -17602.545} C_VEL
LIN {X 0,Y 277.229,Z 252.445,A -85,B 0,C 180,E1 -17606.116,E2 -17606.116} C_VEL
LIN {X 0,Y 277.241,Z 252.449,A -85,B 0,C 180,E1 -17609.55,E2 -17609.55} C_VEL
LIN {X 0,Y 277.335,Z 252.437,A -85,B 0,C 180,E1 -17612.874,E2 -17612.874} C_VEL
LIN {X 0,Y 277.282,Z 252.44,A -85,B 0,C 180,E1 -17616.087,E2 -17616.087} C_VEL
LIN {X 0,Y 277.275,Z 252.444,A -85,B 0,C 180,E1 -17620.773,E2 -17620.773} C_VEL
LIN {X 0,Y 277.386,Z 252.425,A -85,B 0,C 180,E1 -17624.973,E2 -17624.973} C_VEL
LIN {X 0,Y 276.77,Z 252.509,A -85,B 0,C 180,E1 -17626.185,E2 -17626.185} C_VEL
LIN {X 0,Y 273.996,Z 252.858,A -85,B 0,C 180,E1 -17628.161,E2 -17628.161} C_VEL
LIN {X 0,Y 271.622,Z 253.151,A -85,B 0,C 180,E1 -17629.766,E2 -17629.766} C_VEL
LIN {X 0,Y 270.602,Z 253.273,A -85,B 0,C 180,E1 -17631.008,E2 -17631.008} C_VEL
LIN {X 0,Y 270.52,Z 253.28,A -85,B 0,C 180,E1 -17631.429,E2 -17631.429} C_VEL
LIN {X 0,Y 270.515,Z 253.286,A -85,B 0,C 180,E1 -17634.045,E2 -17634.045} C_VEL
LIN {X 0,Y 270.778,Z 253.253,A -85,B 0,C 180,E1 -17638.523,E2 -17638.523} C_VEL
LIN {X 0,Y 270.783,Z 253.248,A -85,B 0,C 180,E1 -17641.497,E2 -17641.497} C_VEL
LIN {X 0,Y 270.575,Z 253.267,A -85,B 0,C 180,E1 -17647.472,E2 -17647.472} C_VEL
LIN {X 0,Y 270.422,Z 253.3,A -85,B 0,C 180,E1 -17650.491,E2 -17650.491} C_VEL
LIN {X 0,Y 270.387,Z 253.299,A -85,B 0,C 180,E1 -17655.075,E2 -17655.075} C_VEL
LIN {X 0,Y 270.244,Z 253.309,A -85,B 0,C 180,E1 -17659.769,E2 -17659.769} C_VEL
LIN {X 0,Y 270.247,Z 253.322,A -85,B 0,C 180,E1 -17664.597,E2 -17664.597} C_VEL
LIN {X 0,Y 270.217,Z 253.315,A -85,B 0,C 180,E1 -17667.924,E2 -17667.924} C_VEL
LIN {X 0,Y 270.194,Z 253.329,A -85,B 0,C 180,E1 -17671.356,E2 -17671.356} C_VEL
LIN {X 0,Y 270.223,Z 253.324,A -85,B 0,C 180,E1 -17674.911,E2 -17674.911} C_VEL
LIN {X 0,Y 270.226,Z 253.322,A -85,B 0,C 180,E1 -17678.715,E2 -17678.715} C_VEL
LIN {X 0,Y 270.142,Z 253.331,A -85,B 0,C 180,E1 -17683.241,E2 -17683.241} C_VEL
LIN {X 0,Y 270.145,Z 253.331,A -85,B 0,C 180,E1 -17687.434,E2 -17687.434} C_VEL
LIN {X 0,Y 270.181,Z 253.331,A -85,B 0,C 180,E1 -17691.367,E2 -17691.367} C_VEL
LIN {X 0,Y 270.226,Z 253.325,A -85,B 0,C 180,E1 -17695.096,E2 -17695.096} C_VEL
LIN {X 0,Y 270.291,Z 253.495,A -85,B 0,C 180,E1 -17697.013,E2 -17697.013} C_VEL
LIN {X 0,Y 272.298,Z 263.161,A -85,B 0,C 180,E1 -17700.631,E2 -17700.631} C_VEL
LIN {X 0,Y 273.292,Z 268.124,A -85,B 0,C 180,E1 -17702.291,E2 -17702.291} C_VEL
LIN {X 0,Y 277.608,Z 281.064,A -85,B 0,C 180,E1 -17703.089,E2 -17703.089} C_VEL
LIN {X 0,Y 281.85,Z 309.937,A -85,B 0,C 180,E1 -17704.316,E2 -17704.316} C_VEL
LIN {X 0,Y 279.653,Z 375.618,A -85,B 0,C 180,E1 -17706.19,E2 -17706.19} C_VEL
LIN {X 0,Y 278.777,Z 389.111,A -85,B 0,C 180,E1 -17706.849,E2 -17706.849} C_VEL
LIN {X 0,Y 277.622,Z 402.066,A -85,B 0,C 180,E1 -17707.779,E2 -17707.779} C_VEL
LIN {X 0,Y 276.218,Z 413.903,A -85,B 0,C 180,E1 -17708.935,E2 -17708.935} C_VEL
LIN {X 0,Y 274.66,Z 425.356,A -85,B 0,C 180,E1 -17710.374,E2 -17710.374} C_VEL
LIN {X 0,Y 273.317,Z 435.738,A -85,B 0,C 180,E1 -17712.025,E2 -17712.025} C_VEL
LIN {X 0,Y 271.963,Z 445.045,A -85,B 0,C 180,E1 -17713.869,E2 -17713.869} C_VEL
LIN {X 0,Y 270.595,Z 454.101,A -85,B 0,C 180,E1 -17716.097,E2 -17716.097} C_VEL
LIN {X 0,Y 269.547,Z 461.348,A -85,B 0,C 180,E1 -17718.34,E2 -17718.34} C_VEL
LIN {X 0,Y 268.758,Z 467.928,A -85,B 0,C 180,E1 -17720.971,E2 -17720.971} C_VEL
LIN {X 0,Y 268.354,Z 472.24,A -85,B 0,C 180,E1 -17723.229,E2 -17723.229} C_VEL
LIN {X 0,Y 268.159,Z 475.441,A -85,B 0,C 180,E1 -17725.488,E2 -17725.488} C_VEL
LIN {X 0,Y 268.144,Z 477.026,A -85,B 0,C 180,E1 -17726.993,E2 -17726.993} C_VEL
LIN {X 0,Y 268.144,Z 478.152,A -85,B 0,C 180,E1 -17728.496,E2 -17728.496} C_VEL
LIN {X 0,Y 268.161,Z 478.846,A -85,B 0,C 180,E1 -17729.997,E2 -17729.997} C_VEL
LIN {X 0,Y 268.143,Z 479.143,A -85,B 0,C 180,E1 -17731.499,E2 -17731.499} C_VEL
LIN {X 0,Y 268.126,Z 479.043,A -85,B 0,C 180,E1 -17733.002,E2 -17733.002} C_VEL
LIN {X 0,Y 268.181,Z 478.144,A -85,B 0,C 180,E1 -17735.166,E2 -17735.166} C_VEL
LIN {X 0,Y 268.564,Z 476.227,A -85,B 0,C 180,E1 -17737.516,E2 -17737.516} C_VEL
LIN {X 0,Y 269.165,Z 473.407,A -85,B 0,C 180,E1 -17739.769,E2 -17739.769} C_VEL
LIN {X 0,Y 270.066,Z 469.566,A -85,B 0,C 180,E1 -17742.013,E2 -17742.013} C_VEL
LIN {X 0,Y 271.316,Z 464.606,A -85,B 0,C 180,E1 -17744.243,E2 -17744.243} C_VEL
LIN {X 0,Y 273.078,Z 458.375,A -85,B 0,C 180,E1 -17746.442,E2 -17746.442} C_VEL
LIN {X 0,Y 275.063,Z 450.969,A -85,B 0,C 180,E1 -17748.536,E2 -17748.536} C_VEL
LIN {X 0,Y 276.954,Z 442.975,A -85,B 0,C 180,E1 -17750.38,E2 -17750.38} C_VEL
LIN {X 0,Y 279.249,Z 433.275,A -85,B 0,C 180,E1 -17752.177,E2 -17752.177} C_VEL
LIN {X 0,Y 281.291,Z 424.044,A -85,B 0,C 180,E1 -17753.56,E2 -17753.56} C_VEL
LIN {X 0,Y 283.424,Z 412.733,A -85,B 0,C 180,E1 -17754.929,E2 -17754.929} C_VEL
LIN {X 0,Y 285.452,Z 400.979,A -85,B 0,C 180,E1 -17756.009,E2 -17756.009} C_VEL
LIN {X 0,Y 287.042,Z 388.306,A -85,B 0,C 180,E1 -17756.881,E2 -17756.881} C_VEL
LIN {X 0,Y 288.331,Z 375.244,A -85,B 0,C 180,E1 -17757.487,E2 -17757.487} C_VEL
LIN {X 0,Y 291.308,Z 312.748,A -85,B 0,C 180,E1 -17759.294,E2 -17759.294} C_VEL
LIN {X 0,Y 288.776,Z 296.661,A -85,B 0,C 180,E1 -17760.259,E2 -17760.259} C_VEL
LIN {X 0,Y 284.43,Z 286.515,A -85,B 0,C 180,E1 -17761.329,E2 -17761.329} C_VEL
LIN {X 0,Y 278.809,Z 275.279,A -85,B 0,C 180,E1 -17762.737,E2 -17762.737} C_VEL
LIN {X 0,Y 275.673,Z 269.717,A -85,B 0,C 180,E1 -17763.539,E2 -17763.539} C_VEL
LIN {X 0,Y 273.921,Z 266.245,A -85,B 0,C 180,E1 -17764.072,E2 -17764.072} C_VEL
LIN {X 0,Y 271.821,Z 258.863,A -85,B 0,C 180,E1 -17767.411,E2 -17767.411} C_VEL
LIN {X 0,Y 270.186,Z 253.488,A -85,B 0,C 180,E1 -17770.189,E2 -17770.189} C_VEL
LIN {X 0,Y 270.159,Z 253.329,A -85,B 0,C 180,E1 -17773.237,E2 -17773.237} C_VEL
LIN {X 0,Y 270.16,Z 253.33,A -85,B 0,C 180,E1 -17777.43,E2 -17777.43} C_VEL
LIN {X 0,Y 270.186,Z 253.325,A -85,B 0,C 180,E1 -17781.361,E2 -17781.361} C_VEL
LIN {X 0,Y 270.203,Z 253.329,A -85,B 0,C 180,E1 -17785.086,E2 -17785.086} C_VEL
LIN {X 0,Y 270.176,Z 253.328,A -85,B 0,C 180,E1 -17789.133,E2 -17789.133} C_VEL
LIN {X 0,Y 270.201,Z 253.329,A -85,B 0,C 180,E1 -17792.165,E2 -17792.165} C_VEL
LIN {X 0,Y 270.229,Z 253.324,A -85,B 0,C 180,E1 -17795.534,E2 -17795.534} C_VEL
LIN {X 0,Y 270.216,Z 253.319,A -85,B 0,C 180,E1 -17800.229,E2 -17800.229} C_VEL
LIN {X 0,Y 270.339,Z 253.303,A -85,B 0,C 180,E1 -17804.923,E2 -17804.923} C_VEL
LIN {X 0,Y 270.377,Z 253.307,A -85,B 0,C 180,E1 -17809.507,E2 -17809.507} C_VEL
LIN {X 0,Y 270.555,Z 253.283,A -85,B 0,C 180,E1 -17812.528,E2 -17812.528} C_VEL
LIN {X 0,Y 270.763,Z 253.258,A -85,B 0,C 180,E1 -17818.503,E2 -17818.503} C_VEL
LIN {X 0,Y 270.768,Z 253.258,A -85,B 0,C 180,E1 -17821.477,E2 -17821.477} C_VEL
LIN {X 0,Y 270.582,Z 253.28,A -85,B 0,C 180,E1 -17827.452,E2 -17827.452} C_VEL
LIN {X 0,Y 270.569,Z 253.514,A -85,B 0,C 180,E1 -17828.203,E2 -17828.203} C_VEL
LIN {X 0,Y 272.502,Z 260.539,A -85,B 0,C 180,E1 -17831.604,E2 -17831.604} C_VEL
LIN {X 0,Y 273.323,Z 262.373,A -85,B 0,C 180,E1 -17831.954,E2 -17831.954} C_VEL
LIN {X 0,Y 278.278,Z 270.584,A -85,B 0,C 180,E1 -17833.244,E2 -17833.244} C_VEL
LIN {X 0,Y 284.365,Z 282.065,A -85,B 0,C 180,E1 -17834.755,E2 -17834.755} C_VEL
LIN {X 0,Y 289.991,Z 294.542,A -85,B 0,C 180,E1 -17836.112,E2 -17836.112} C_VEL
LIN {X 0,Y 291.183,Z 297.986,A -85,B 0,C 180,E1 -17836.418,E2 -17836.418} C_VEL
LIN {X 0,Y 291.762,Z 302.135,A -85,B 0,C 180,E1 -17836.654,E2 -17836.654} C_VEL
LIN {X 0,Y 288.442,Z 369.337,A -85,B 0,C 180,E1 -17838.594,E2 -17838.594} C_VEL
LIN {X 0,Y 287.141,Z 383.115,A -85,B 0,C 180,E1 -17839.26,E2 -17839.26} C_VEL
LIN {X 0,Y 285.599,Z 395.446,A -85,B 0,C 180,E1 -17840.141,E2 -17840.141} C_VEL
LIN {X 0,Y 283.712,Z 407.299,A -85,B 0,C 180,E1 -17841.285,E2 -17841.285} C_VEL
LIN {X 0,Y 281.486,Z 418.903,A -85,B 0,C 180,E1 -17842.726,E2 -17842.726} C_VEL
LIN {X 0,Y 279.07,Z 429.794,A -85,B 0,C 180,E1 -17844.461,E2 -17844.461} C_VEL
LIN {X 0,Y 276.715,Z 439.333,A -85,B 0,C 180,E1 -17846.376,E2 -17846.376} C_VEL
LIN {X 0,Y 274.379,Z 448.408,A -85,B 0,C 180,E1 -17848.69,E2 -17848.69} C_VEL
LIN {X 0,Y 272.313,Z 455.695,A -85,B 0,C 180,E1 -17851.062,E2 -17851.062} C_VEL
LIN {X 0,Y 271.079,Z 460.338,A -85,B 0,C 180,E1 -17852.973,E2 -17852.973} C_VEL
LIN {X 0,Y 270.076,Z 464.142,A -85,B 0,C 180,E1 -17854.909,E2 -17854.909} C_VEL
LIN {X 0,Y 269.253,Z 467.164,A -85,B 0,C 180,E1 -17856.879,E2 -17856.879} C_VEL
LIN {X 0,Y 268.602,Z 469.412,A -85,B 0,C 180,E1 -17858.884,E2 -17858.884} C_VEL
LIN {X 0,Y 268.163,Z 470.941,A -85,B 0,C 180,E1 -17860.918,E2 -17860.918} C_VEL
LIN {X 0,Y 267.917,Z 471.746,A -85,B 0,C 180,E1 -17862.985,E2 -17862.985} C_VEL
LIN {X 0,Y 267.771,Z 471.743,A -85,B 0,C 180,E1 -17865.107,E2 -17865.107} C_VEL
LIN {X 0,Y 267.742,Z 470.898,A -85,B 0,C 180,E1 -17867.286,E2 -17867.286} C_VEL
LIN {X 0,Y 267.864,Z 469.134,A -85,B 0,C 180,E1 -17869.522,E2 -17869.522} C_VEL
LIN {X 0,Y 268.208,Z 466.346,A -85,B 0,C 180,E1 -17871.802,E2 -17871.802} C_VEL
LIN {X 0,Y 268.709,Z 462.344,A -85,B 0,C 180,E1 -17874.151,E2 -17874.151} C_VEL
LIN {X 0,Y 269.469,Z 456.33,A -85,B 0,C 180,E1 -17876.794,E2 -17876.794} C_VEL
LIN {X 0,Y 270.371,Z 449.671,A -85,B 0,C 180,E1 -17879.045,E2 -17879.045} C_VEL
LIN {X 0,Y 271.482,Z 442.266,A -85,B 0,C 180,E1 -17881.062,E2 -17881.062} C_VEL
LIN {X 0,Y 272.95,Z 432.425,A -85,B 0,C 180,E1 -17883.222,E2 -17883.222} C_VEL
LIN {X 0,Y 274.47,Z 422.1,A -85,B 0,C 180,E1 -17885.011,E2 -17885.011} C_VEL
LIN {X 0,Y 275.939,Z 410.647,A -85,B 0,C 180,E1 -17886.595,E2 -17886.595} C_VEL
LIN {X 0,Y 277.288,Z 399.3,A -85,B 0,C 180,E1 -17887.821,E2 -17887.821} C_VEL
LIN {X 0,Y 278.459,Z 386.182,A -85,B 0,C 180,E1 -17888.889,E2 -17888.889} C_VEL
LIN {X 0,Y 279.452,Z 372.769,A -85,B 0,C 180,E1 -17889.652,E2 -17889.652} C_VEL
LIN {X 0,Y 280.147,Z 356.18,A -85,B 0,C 180,E1 -17890.207,E2 -17890.207} C_VEL
LIN {X 0,Y 281.971,Z 296.843,A -85,B 0,C 180,E1 -17891.886,E2 -17891.886} C_VEL
LIN {X 0,Y 279.479,Z 282.766,A -85,B 0,C 180,E1 -17892.518,E2 -17892.518} C_VEL
LIN {X 0,Y 271.881,Z 261.134,A -85,B 0,C 180,E1 -17893.869,E2 -17893.869} C_VEL
LIN {X 0,Y 271.617,Z 259.808,A -85,B 0,C 180,E1 -17894.238,E2 -17894.238} C_VEL
LIN {X 0,Y 270.39,Z 253.617,A -85,B 0,C 180,E1 -17896.666,E2 -17896.666} C_VEL
LIN {X 0,Y 270.317,Z 253.315,A -85,B 0,C 180,E1 -17897.235,E2 -17897.235} C_VEL
LIN {X 0,Y 270.494,Z 253.292,A -85,B 0,C 180,E1 -17901.034,E2 -17901.034} C_VEL
LIN {X 0,Y 270.475,Z 253.292,A -85,B 0,C 180,E1 -17904.037,E2 -17904.037} C_VEL
LIN {X 0,Y 270.726,Z 253.262,A -85,B 0,C 180,E1 -17908.515,E2 -17908.515} C_VEL
LIN {X 0,Y 270.727,Z 253.262,A -85,B 0,C 180,E1 -17911.49,E2 -17911.49} C_VEL
LIN {X 0,Y 270.541,Z 253.285,A -85,B 0,C 180,E1 -17917.466,E2 -17917.466} C_VEL
LIN {X 0,Y 270.379,Z 253.295,A -85,B 0,C 180,E1 -17920.486,E2 -17920.486} C_VEL
LIN {X 0,Y 270.322,Z 253.312,A -85,B 0,C 180,E1 -17925.072,E2 -17925.072} C_VEL
LIN {X 0,Y 270.242,Z 253.316,A -85,B 0,C 180,E1 -17929.762,E2 -17929.762} C_VEL
LIN {X 0,Y 270.184,Z 253.326,A -85,B 0,C 180,E1 -17934.597,E2 -17934.597} C_VEL
LIN {X 0,Y 270.219,Z 253.311,A -85,B 0,C 180,E1 -17937.917,E2 -17937.917} C_VEL
LIN {X 0,Y 270.136,Z 253.326,A -85,B 0,C 180,E1 -17941.357,E2 -17941.357} C_VEL
LIN {X 0,Y 270.168,Z 253.329,A -85,B 0,C 180,E1 -17944.913,E2 -17944.913} C_VEL
LIN {X 0,Y 270.181,Z 253.325,A -85,B 0,C 180,E1 -17948.727,E2 -17948.727} C_VEL
LIN {X 0,Y 270.191,Z 253.33,A -85,B 0,C 180,E1 -17952.557,E2 -17952.557} C_VEL
LIN {X 0,Y 270.197,Z 253.324,A -85,B 0,C 180,E1 -17956.747,E2 -17956.747} C_VEL
LIN {X 0,Y 270.217,Z 253.322,A -85,B 0,C 180,E1 -17959.458,E2 -17959.458} C_VEL
LIN {X 0,Y 270.231,Z 253.318,A -85,B 0,C 180,E1 -17963.732,E2 -17963.732} C_VEL
LIN {X 0,Y 270.18,Z 253.327,A -85,B 0,C 180,E1 -17966.904,E2 -17966.904} C_VEL
LIN {X 0,Y 270.174,Z 253.329,A -85,B 0,C 180,E1 -17970.394,E2 -17970.394} C_VEL
LIN {X 0,Y 270.241,Z 253.314,A -85,B 0,C 180,E1 -17973.774,E2 -17973.774} C_VEL
LIN {X 0,Y 270.194,Z 253.326,A -85,B 0,C 180,E1 -17977.048,E2 -17977.048} C_VEL
LIN {X 0,Y 270.214,Z 253.323,A -85,B 0,C 180,E1 -17980.25,E2 -17980.25} C_VEL
LIN {X 0,Y 270.362,Z 253.3,A -85,B 0,C 180,E1 -17984.95,E2 -17984.95} C_VEL
LIN {X 0,Y 270.411,Z 253.302,A -85,B 0,C 180,E1 -17989.528,E2 -17989.528} C_VEL
LIN {X 0,Y 270.52,Z 253.28,A -85,B 0,C 180,E1 -17991.429,E2 -17991.429} C_VEL
LIN {X 0,Y 269.838,Z 253.364,A -85,B 0,C 180,E1 -17992.671,E2 -17992.671} C_VEL
LIN {X 0,Y 266.953,Z 253.727,A -85,B 0,C 180,E1 -17994.693,E2 -17994.693} C_VEL
LIN {X 0,Y 264.585,Z 254.026,A -85,B 0,C 180,E1 -17996.338,E2 -17996.338} C_VEL
LIN {X 0,Y 263.678,Z 254.14,A -85,B 0,C 180,E1 -17997.613,E2 -17997.613} C_VEL
LIN {X 0,Y 263.661,Z 254.137,A -85,B 0,C 180,E1 -17998.044,E2 -17998.044} C_VEL
LIN {X 0,Y 263.746,Z 254.125,A -85,B 0,C 180,E1 -18001.537,E2 -18001.537} C_VEL
LIN {X 0,Y 263.54,Z 254.143,A -85,B 0,C 180,E1 -18007.672,E2 -18007.672} C_VEL
LIN {X 0,Y 263.362,Z 254.179,A -85,B 0,C 180,E1 -18010.776,E2 -18010.776} C_VEL
LIN {X 0,Y 263.329,Z 254.177,A -85,B 0,C 180,E1 -18015.489,E2 -18015.489} C_VEL
LIN {X 0,Y 263.23,Z 254.184,A -85,B 0,C 180,E1 -18020.319,E2 -18020.319} C_VEL
LIN {X 0,Y 263.19,Z 254.199,A -85,B 0,C 180,E1 -18025.302,E2 -18025.302} C_VEL
LIN {X 0,Y 263.147,Z 254.196,A -85,B 0,C 180,E1 -18028.743,E2 -18028.743} C_VEL
LIN {X 0,Y 263.152,Z 254.203,A -85,B 0,C 180,E1 -18032.295,E2 -18032.295} C_VEL
LIN {X 0,Y 263.181,Z 254.191,A -85,B 0,C 180,E1 -18035.988,E2 -18035.988} C_VEL
LIN {X 0,Y 263.115,Z 254.209,A -85,B 0,C 180,E1 -18039.881,E2 -18039.881} C_VEL
LIN {X 0,Y 263.094,Z 254.213,A -85,B 0,C 180,E1 -18044,E2 -18044} C_VEL
LIN {X 0,Y 263.088,Z 254.213,A -85,B 0,C 180,E1 -18048.426,E2 -18048.426} C_VEL
LIN {X 0,Y 263.132,Z 254.209,A -85,B 0,C 180,E1 -18052.096,E2 -18052.096} C_VEL
LIN {X 0,Y 263.225,Z 254.242,A -85,B 0,C 180,E1 -18056.469,E2 -18056.469} C_VEL
LIN {X 0,Y 263.874,Z 257.449,A -85,B 0,C 180,E1 -18057.811,E2 -18057.811} C_VEL
LIN {X 0,Y 265.979,Z 267.73,A -85,B 0,C 180,E1 -18061.613,E2 -18061.613} C_VEL
LIN {X 0,Y 268.367,Z 274.667,A -85,B 0,C 180,E1 -18062.112,E2 -18062.112} C_VEL
LIN {X 0,Y 271.144,Z 283.096,A -85,B 0,C 180,E1 -18062.616,E2 -18062.616} C_VEL
LIN {X 0,Y 275.133,Z 311.295,A -85,B 0,C 180,E1 -18063.846,E2 -18063.846} C_VEL
LIN {X 0,Y 272.926,Z 375.318,A -85,B 0,C 180,E1 -18065.717,E2 -18065.717} C_VEL
LIN {X 0,Y 272.048,Z 388.871,A -85,B 0,C 180,E1 -18066.393,E2 -18066.393} C_VEL
LIN {X 0,Y 270.906,Z 401.314,A -85,B 0,C 180,E1 -18067.298,E2 -18067.298} C_VEL
LIN {X 0,Y 269.551,Z 412.532,A -85,B 0,C 180,E1 -18068.388,E2 -18068.388} C_VEL
LIN {X 0,Y 267.922,Z 424.213,A -85,B 0,C 180,E1 -18069.859,E2 -18069.859} C_VEL
LIN {X 0,Y 266.487,Z 434.788,A -85,B 0,C 180,E1 -18071.548,E2 -18071.548} C_VEL
LIN {X 0,Y 265.125,Z 444.291,A -85,B 0,C 180,E1 -18073.441,E2 -18073.441} C_VEL
LIN {X 0,Y 263.648,Z 453.456,A -85,B 0,C 180,E1 -18075.723,E2 -18075.723} C_VEL
LIN {X 0,Y 262.526,Z 460.825,A -85,B 0,C 180,E1 -18078.023,E2 -18078.023} C_VEL
LIN {X 0,Y 261.921,Z 465.786,A -85,B 0,C 180,E1 -18079.953,E2 -18079.953} C_VEL
LIN {X 0,Y 261.389,Z 470.578,A -85,B 0,C 180,E1 -18082.271,E2 -18082.271} C_VEL
LIN {X 0,Y 261.114,Z 474.57,A -85,B 0,C 180,E1 -18084.861,E2 -18084.861} C_VEL
LIN {X 0,Y 261.043,Z 476.781,A -85,B 0,C 180,E1 -18086.911,E2 -18086.911} C_VEL
LIN {X 0,Y 261.053,Z 477.969,A -85,B 0,C 180,E1 -18088.455,E2 -18088.455} C_VEL
LIN {X 0,Y 261.09,Z 478.698,A -85,B 0,C 180,E1 -18089.997,E2 -18089.997} C_VEL
LIN {X 0,Y 261.051,Z 479.026,A -85,B 0,C 180,E1 -18091.54,E2 -18091.54} C_VEL
LIN {X 0,Y 261.026,Z 478.96,A -85,B 0,C 180,E1 -18093.084,E2 -18093.084} C_VEL
LIN {X 0,Y 261.074,Z 478.272,A -85,B 0,C 180,E1 -18095.042,E2 -18095.042} C_VEL
LIN {X 0,Y 261.527,Z 476.28,A -85,B 0,C 180,E1 -18097.719,E2 -18097.719} C_VEL
LIN {X 0,Y 262.149,Z 473.53,A -85,B 0,C 180,E1 -18100.033,E2 -18100.033} C_VEL
LIN {X 0,Y 263.127,Z 469.76,A -85,B 0,C 180,E1 -18102.335,E2 -18102.335} C_VEL
LIN {X 0,Y 264.447,Z 464.877,A -85,B 0,C 180,E1 -18104.621,E2 -18104.621} C_VEL
LIN {X 0,Y 266.291,Z 458.758,A -85,B 0,C 180,E1 -18106.874,E2 -18106.874} C_VEL
LIN {X 0,Y 268.583,Z 450.611,A -85,B 0,C 180,E1 -18109.251,E2 -18109.251} C_VEL
LIN {X 0,Y 270.79,Z 441.744,A -85,B 0,C 180,E1 -18111.303,E2 -18111.303} C_VEL
LIN {X 0,Y 273.445,Z 430.967,A -85,B 0,C 180,E1 -18113.273,E2 -18113.273} C_VEL
LIN {X 0,Y 275.984,Z 419.868,A -85,B 0,C 180,E1 -18114.843,E2 -18114.843} C_VEL
LIN {X 0,Y 278.012,Z 409.134,A -85,B 0,C 180,E1 -18116.052,E2 -18116.052} C_VEL
LIN {X 0,Y 280.084,Z 396.362,A -85,B 0,C 180,E1 -18117.15,E2 -18117.15} C_VEL
LIN {X 0,Y 281.636,Z 384.26,A -85,B 0,C 180,E1 -18117.894,E2 -18117.894} C_VEL
LIN {X 0,Y 282.826,Z 370.672,A -85,B 0,C 180,E1 -18118.444,E2 -18118.444} C_VEL
LIN {X 0,Y 285.567,Z 313.573,A -85,B 0,C 180,E1 -18120.129,E2 -18120.129} C_VEL
LIN {X 0,Y 283.335,Z 299.39,A -85,B 0,C 180,E1 -18121.017,E2 -18121.017} C_VEL
LIN {X 0,Y 278.808,Z 288.872,A -85,B 0,C 180,E1 -18122.191,E2 -18122.191} C_VEL
LIN {X 0,Y 273.37,Z 278.177,A -85,B 0,C 180,E1 -18123.625,E2 -18123.625} C_VEL
LIN {X 0,Y 268.993,Z 270.298,A -85,B 0,C 180,E1 -18124.842,E2 -18124.842} C_VEL
LIN {X 0,Y 266.664,Z 266.107,A -85,B 0,C 180,E1 -18125.569,E2 -18125.569} C_VEL
LIN {X 0,Y 264.879,Z 259.935,A -85,B 0,C 180,E1 -18128.531,E2 -18128.531} C_VEL
LIN {X 0,Y 263.095,Z 254.242,A -85,B 0,C 180,E1 -18131.784,E2 -18131.784} C_VEL
LIN {X 0,Y 263.089,Z 254.211,A -85,B 0,C 180,E1 -18136.154,E2 -18136.154} C_VEL
LIN {X 0,Y 263.122,Z 254.203,A -85,B 0,C 180,E1 -18140.763,E2 -18140.763} C_VEL
LIN {X 0,Y 263.162,Z 254.197,A -85,B 0,C 180,E1 -18144.008,E2 -18144.008} C_VEL
LIN {X 0,Y 263.132,Z 254.204,A -85,B 0,C 180,E1 -18147.702,E2 -18147.702} C_VEL
LIN {X 0,Y 263.146,Z 254.207,A -85,B 0,C 180,E1 -18151.799,E2 -18151.799} C_VEL
LIN {X 0,Y 263.191,Z 254.202,A -85,B 0,C 180,E1 -18155.209,E2 -18155.209} C_VEL
LIN {X 0,Y 263.206,Z 254.197,A -85,B 0,C 180,E1 -18159.679,E2 -18159.679} C_VEL
LIN {X 0,Y 263.286,Z 254.18,A -85,B 0,C 180,E1 -18164.509,E2 -18164.509} C_VEL
LIN {X 0,Y 263.322,Z 254.184,A -85,B 0,C 180,E1 -18169.223,E2 -18169.223} C_VEL
LIN {X 0,Y 263.519,Z 254.159,A -85,B 0,C 180,E1 -18172.327,E2 -18172.327} C_VEL
LIN {X 0,Y 263.726,Z 254.135,A -85,B 0,C 180,E1 -18178.463,E2 -18178.463} C_VEL
LIN {X 0,Y 263.732,Z 254.134,A -85,B 0,C 180,E1 -18181.517,E2 -18181.517} C_VEL
LIN {X 0,Y 263.506,Z 254.3,A -85,B 0,C 180,E1 -18186.69,E2 -18186.69} C_VEL
LIN {X 0,Y 264.889,Z 258.779,A -85,B 0,C 180,E1 -18189.149,E2 -18189.149} C_VEL
LIN {X 0,Y 265.518,Z 261.182,A -85,B 0,C 180,E1 -18190.233,E2 -18190.233} C_VEL
LIN {X 0,Y 269.909,Z 268.571,A -85,B 0,C 180,E1 -18191.536,E2 -18191.536} C_VEL
LIN {X 0,Y 275.15,Z 277.609,A -85,B 0,C 180,E1 -18192.951,E2 -18192.951} C_VEL
LIN {X 0,Y 281.176,Z 289.573,A -85,B 0,C 180,E1 -18194.515,E2 -18194.515} C_VEL
LIN {X 0,Y 285.652,Z 300.209,A -85,B 0,C 180,E1 -18195.646,E2 -18195.646} C_VEL
LIN {X 0,Y 286.049,Z 303.478,A -85,B 0,C 180,E1 -18195.83,E2 -18195.83} C_VEL
LIN {X 0,Y 282.612,Z 369.433,A -85,B 0,C 180,E1 -18197.781,E2 -18197.781} C_VEL
LIN {X 0,Y 281.23,Z 383.367,A -85,B 0,C 180,E1 -18198.47,E2 -18198.47} C_VEL
LIN {X 0,Y 279.657,Z 395.349,A -85,B 0,C 180,E1 -18199.343,E2 -18199.343} C_VEL
LIN {X 0,Y 277.451,Z 408.522,A -85,B 0,C 180,E1 -18200.652,E2 -18200.652} C_VEL
LIN {X 0,Y 275.094,Z 419.973,A -85,B 0,C 180,E1 -18202.125,E2 -18202.125} C_VEL
LIN {X 0,Y 272.836,Z 429.709,A -85,B 0,C 180,E1 -18203.721,E2 -18203.721} C_VEL
LIN {X 0,Y 270.475,Z 438.721,A -85,B 0,C 180,E1 -18205.543,E2 -18205.543} C_VEL
LIN {X 0,Y 268.256,Z 446.969,A -85,B 0,C 180,E1 -18207.625,E2 -18207.625} C_VEL
LIN {X 0,Y 266.464,Z 453.024,A -85,B 0,C 180,E1 -18209.504,E2 -18209.504} C_VEL
LIN {X 0,Y 264.525,Z 459.63,A -85,B 0,C 180,E1 -18212.084,E2 -18212.084} C_VEL
LIN {X 0,Y 263.328,Z 463.784,A -85,B 0,C 180,E1 -18214.177,E2 -18214.177} C_VEL
LIN {X 0,Y 262.281,Z 467.314,A -85,B 0,C 180,E1 -18216.504,E2 -18216.504} C_VEL
LIN {X 0,Y 261.539,Z 469.78,A -85,B 0,C 180,E1 -18218.811,E2 -18218.811} C_VEL
LIN {X 0,Y 261.049,Z 471.283,A -85,B 0,C 180,E1 -18221.083,E2 -18221.083} C_VEL
LIN {X 0,Y 260.779,Z 471.905,A -85,B 0,C 180,E1 -18223.315,E2 -18223.315} C_VEL
LIN {X 0,Y 260.658,Z 471.709,A -85,B 0,C 180,E1 -18225.495,E2 -18225.495} C_VEL
LIN {X 0,Y 260.638,Z 470.747,A -85,B 0,C 180,E1 -18227.619,E2 -18227.619} C_VEL
LIN {X 0,Y 260.779,Z 468.999,A -85,B 0,C 180,E1 -18229.703,E2 -18229.703} C_VEL
LIN {X 0,Y 261.094,Z 466.519,A -85,B 0,C 180,E1 -18231.753,E2 -18231.753} C_VEL
LIN {X 0,Y 261.503,Z 463.319,A -85,B 0,C 180,E1 -18233.757,E2 -18233.757} C_VEL
LIN {X 0,Y 262.159,Z 458.253,A -85,B 0,C 180,E1 -18236.183,E2 -18236.183} C_VEL
LIN {X 0,Y 263.128,Z 451.467,A -85,B 0,C 180,E1 -18238.701,E2 -18238.701} C_VEL
LIN {X 0,Y 264.257,Z 443.946,A -85,B 0,C 180,E1 -18240.913,E2 -18240.913} C_VEL
LIN {X 0,Y 265.636,Z 434.771,A -85,B 0,C 180,E1 -18243.062,E2 -18243.062} C_VEL
LIN {X 0,Y 267.124,Z 425.006,A -85,B 0,C 180,E1 -18244.903,E2 -18244.903} C_VEL
LIN {X 0,Y 268.625,Z 414.891,A -85,B 0,C 180,E1 -18246.44,E2 -18246.44} C_VEL
LIN {X 0,Y 269.997,Z 403.402,A -85,B 0,C 180,E1 -18247.828,E2 -18247.828} C_VEL
LIN {X 0,Y 271.315,Z 390.888,A -85,B 0,C 180,E1 -18248.986,E2 -18248.986} C_VEL
LIN {X 0,Y 272.343,Z 377.861,A -85,B 0,C 180,E1 -18249.861,E2 -18249.861} C_VEL
LIN {X 0,Y 273.174,Z 363.64,A -85,B 0,C 180,E1 -18250.464,E2 -18250.464} C_VEL
LIN {X 0,Y 275.317,Z 297.748,A -85,B 0,C 180,E1 -18252.377,E2 -18252.377} C_VEL
LIN {X 0,Y 272.941,Z 284.582,A -85,B 0,C 180,E1 -18252.987,E2 -18252.987} C_VEL
LIN {X 0,Y 264.687,Z 261.152,A -85,B 0,C 180,E1 -18254.506,E2 -18254.506} C_VEL
LIN {X 0,Y 263.801,Z 256.795,A -85,B 0,C 180,E1 -18256.13,E2 -18256.13} C_VEL
LIN {X 0,Y 263.295,Z 254.216,A -85,B 0,C 180,E1 -18257.281,E2 -18257.281} C_VEL
LIN {X 0,Y 263.455,Z 254.17,A -85,B 0,C 180,E1 -18260.793,E2 -18260.793} C_VEL
LIN {X 0,Y 263.447,Z 254.168,A -85,B 0,C 180,E1 -18263.877,E2 -18263.877} C_VEL
LIN {X 0,Y 263.692,Z 254.138,A -85,B 0,C 180,E1 -18268.475,E2 -18268.475} C_VEL
LIN {X 0,Y 263.692,Z 254.138,A -85,B 0,C 180,E1 -18271.53,E2 -18271.53} C_VEL
LIN {X 0,Y 263.503,Z 254.161,A -85,B 0,C 180,E1 -18277.666,E2 -18277.666} C_VEL
LIN {X 0,Y 263.309,Z 254.176,A -85,B 0,C 180,E1 -18280.771,E2 -18280.771} C_VEL
LIN {X 0,Y 263.269,Z 254.19,A -85,B 0,C 180,E1 -18285.485,E2 -18285.485} C_VEL
LIN {X 0,Y 263.206,Z 254.194,A -85,B 0,C 180,E1 -18290.314,E2 -18290.314} C_VEL
LIN {X 0,Y 263.139,Z 254.204,A -85,B 0,C 180,E1 -18295.301,E2 -18295.301} C_VEL
LIN {X 0,Y 263.116,Z 254.189,A -85,B 0,C 180,E1 -18298.74,E2 -18298.74} C_VEL
LIN {X 0,Y 263.086,Z 254.211,A -85,B 0,C 180,E1 -18302.297,E2 -18302.297} C_VEL
LIN {X 0,Y 263.142,Z 254.208,A -85,B 0,C 180,E1 -18305.988,E2 -18305.988} C_VEL
LIN {X 0,Y 263.119,Z 254.204,A -85,B 0,C 180,E1 -18309.873,E2 -18309.873} C_VEL
LIN {X 0,Y 263.154,Z 254.204,A -85,B 0,C 180,E1 -18313.98,E2 -18313.98} C_VEL
LIN {X 0,Y 263.18,Z 254.198,A -85,B 0,C 180,E1 -18318.396,E2 -18318.396} C_VEL
LIN {X 0,Y 263.161,Z 254.202,A -85,B 0,C 180,E1 -18322.119,E2 -18322.119} C_VEL
LIN {X 0,Y 263.16,Z 254.196,A -85,B 0,C 180,E1 -18325.902,E2 -18325.902} C_VEL
LIN {X 0,Y 263.119,Z 254.208,A -85,B 0,C 180,E1 -18329.517,E2 -18329.517} C_VEL
LIN {X 0,Y 263.172,Z 254.201,A -85,B 0,C 180,E1 -18333.014,E2 -18333.014} C_VEL
LIN {X 0,Y 263.138,Z 254.201,A -85,B 0,C 180,E1 -18336.395,E2 -18336.395} C_VEL
LIN {X 0,Y 263.199,Z 254.199,A -85,B 0,C 180,E1 -18339.7,E2 -18339.7} C_VEL
LIN {X 0,Y 263.304,Z 254.178,A -85,B 0,C 180,E1 -18344.531,E2 -18344.531} C_VEL
LIN {X 0,Y 263.353,Z 254.179,A -85,B 0,C 180,E1 -18349.245,E2 -18349.245} C_VEL
LIN {X 0,Y 263.528,Z 254.15,A -85,B 0,C 180,E1 -18352.348,E2 -18352.348} C_VEL
LIN {X 0,Y 263.661,Z 254.137,A -85,B 0,C 180,E1 -18358.044,E2 -18358.044} C_VEL
LIN {X 0,Y 263.097,Z 254.211,A -85,B 0,C 180,E1 -18359.319,E2 -18359.319} C_VEL
LIN {X 0,Y 261.463,Z 254.412,A -85,B 0,C 180,E1 -18360.568,E2 -18360.568} C_VEL
LIN {X 0,Y 257.486,Z 254.895,A -85,B 0,C 180,E1 -18363.077,E2 -18363.077} C_VEL
LIN {X 0,Y 256.385,Z 255.024,A -85,B 0,C 180,E1 -18364.392,E2 -18364.392} C_VEL
LIN {X 0,Y 256.314,Z 255.029,A -85,B 0,C 180,E1 -18364.838,E2 -18364.838} C_VEL
LIN {X 0,Y 256.482,Z 255.022,A -85,B 0,C 180,E1 -18367.885,E2 -18367.885} C_VEL
LIN {X 0,Y 256.303,Z 255.056,A -85,B 0,C 180,E1 -18371.076,E2 -18371.076} C_VEL
LIN {X 0,Y 256.25,Z 255.059,A -85,B 0,C 180,E1 -18375.928,E2 -18375.928} C_VEL
LIN {X 0,Y 256.143,Z 255.073,A -85,B 0,C 180,E1 -18381.106,E2 -18381.106} C_VEL
LIN {X 0,Y 256.156,Z 255.076,A -85,B 0,C 180,E1 -18385.118,E2 -18385.118} C_VEL
LIN {X 0,Y 256.068,Z 255.08,A -85,B 0,C 180,E1 -18389.615,E2 -18389.615} C_VEL
LIN {X 0,Y 256.092,Z 255.086,A -85,B 0,C 180,E1 -18393.299,E2 -18393.299} C_VEL
LIN {X 0,Y 256.144,Z 255.071,A -85,B 0,C 180,E1 -18397.276,E2 -18397.276} C_VEL
LIN {X 0,Y 256.034,Z 255.09,A -85,B 0,C 180,E1 -18401.218,E2 -18401.218} C_VEL
LIN {X 0,Y 256.037,Z 255.091,A -85,B 0,C 180,E1 -18405.546,E2 -18405.546} C_VEL
LIN {X 0,Y 256.053,Z 255.09,A -85,B 0,C 180,E1 -18410.233,E2 -18410.233} C_VEL
LIN {X 0,Y 256.13,Z 255.081,A -85,B 0,C 180,E1 -18412.865,E2 -18412.865} C_VEL
LIN {X 0,Y 256.177,Z 255.299,A -85,B 0,C 180,E1 -18416.173,E2 -18416.173} C_VEL
LIN {X 0,Y 258.453,Z 266.242,A -85,B 0,C 180,E1 -18420.491,E2 -18420.491} C_VEL
LIN {X 0,Y 258.79,Z 267.873,A -85,B 0,C 180,E1 -18420.991,E2 -18420.991} C_VEL
LIN {X 0,Y 264.623,Z 284.731,A -85,B 0,C 180,E1 -18422.128,E2 -18422.128} C_VEL
LIN {X 0,Y 268.472,Z 311.636,A -85,B 0,C 180,E1 -18423.328,E2 -18423.328} C_VEL
LIN {X 0,Y 266.161,Z 375.831,A -85,B 0,C 180,E1 -18425.267,E2 -18425.267} C_VEL
LIN {X 0,Y 265.261,Z 389.17,A -85,B 0,C 180,E1 -18425.959,E2 -18425.959} C_VEL
LIN {X 0,Y 264.102,Z 401.504,A -85,B 0,C 180,E1 -18426.887,E2 -18426.887} C_VEL
LIN {X 0,Y 262.697,Z 412.632,A -85,B 0,C 180,E1 -18428.001,E2 -18428.001} C_VEL
LIN {X 0,Y 261.022,Z 424.27,A -85,B 0,C 180,E1 -18429.509,E2 -18429.509} C_VEL
LIN {X 0,Y 259.486,Z 435.255,A -85,B 0,C 180,E1 -18431.319,E2 -18431.319} C_VEL
LIN {X 0,Y 257.983,Z 445.122,A -85,B 0,C 180,E1 -18433.376,E2 -18433.376} C_VEL
LIN {X 0,Y 256.513,Z 454.134,A -85,B 0,C 180,E1 -18435.722,E2 -18435.722} C_VEL
LIN {X 0,Y 255.397,Z 461.325,A -85,B 0,C 180,E1 -18438.087,E2 -18438.087} C_VEL
LIN {X 0,Y 254.683,Z 467.047,A -85,B 0,C 180,E1 -18440.467,E2 -18440.467} C_VEL
LIN {X 0,Y 254.203,Z 471.517,A -85,B 0,C 180,E1 -18442.851,E2 -18442.851} C_VEL
LIN {X 0,Y 254.003,Z 474.866,A -85,B 0,C 180,E1 -18445.236,E2 -18445.236} C_VEL
LIN {X 0,Y 253.947,Z 476.519,A -85,B 0,C 180,E1 -18446.824,E2 -18446.824} C_VEL
LIN {X 0,Y 253.963,Z 477.756,A -85,B 0,C 180,E1 -18448.412,E2 -18448.412} C_VEL
LIN {X 0,Y 253.998,Z 478.545,A -85,B 0,C 180,E1 -18449.997,E2 -18449.997} C_VEL
LIN {X 0,Y 253.961,Z 478.908,A -85,B 0,C 180,E1 -18451.583,E2 -18451.583} C_VEL
LIN {X 0,Y 253.93,Z 478.876,A -85,B 0,C 180,E1 -18453.17,E2 -18453.17} C_VEL
LIN {X 0,Y 253.979,Z 478.384,A -85,B 0,C 180,E1 -18454.938,E2 -18454.938} C_VEL
LIN {X 0,Y 254.465,Z 476.333,A -85,B 0,C 180,E1 -18457.935,E2 -18457.935} C_VEL
LIN {X 0,Y 255.452,Z 472.571,A -85,B 0,C 180,E1 -18461.101,E2 -18461.101} C_VEL
LIN {X 0,Y 256.602,Z 468.537,A -85,B 0,C 180,E1 -18463.459,E2 -18463.459} C_VEL
LIN {X 0,Y 258.5,Z 462.36,A -85,B 0,C 180,E1 -18466.178,E2 -18466.178} C_VEL
LIN {X 0,Y 260.657,Z 455.638,A -85,B 0,C 180,E1 -18468.467,E2 -18468.467} C_VEL
LIN {X 0,Y 262.879,Z 447.504,A -85,B 0,C 180,E1 -18470.702,E2 -18470.702} C_VEL
LIN {X 0,Y 265.217,Z 438.882,A -85,B 0,C 180,E1 -18472.593,E2 -18472.593} C_VEL
LIN {X 0,Y 267.861,Z 428.514,A -85,B 0,C 180,E1 -18474.405,E2 -18474.405} C_VEL
LIN {X 0,Y 270.491,Z 416.959,A -85,B 0,C 180,E1 -18476.002,E2 -18476.002} C_VEL
LIN {X 0,Y 272.766,Z 405.519,A -85,B 0,C 180,E1 -18477.212,E2 -18477.212} C_VEL
LIN {X 0,Y 274.753,Z 392.702,A -85,B 0,C 180,E1 -18478.24,E2 -18478.24} C_VEL
LIN {X 0,Y 276.372,Z 379.572,A -85,B 0,C 180,E1 -18478.97,E2 -18478.97} C_VEL
LIN {X 0,Y 277.475,Z 363.246,A -85,B 0,C 180,E1 -18479.531,E2 -18479.531} C_VEL
LIN {X 0,Y 279.922,Z 314.682,A -85,B 0,C 180,E1 -18480.987,E2 -18480.987} C_VEL
LIN {X 0,Y 277.993,Z 302.296,A -85,B 0,C 180,E1 -18481.798,E2 -18481.798} C_VEL
LIN {X 0,Y 273.461,Z 291.621,A -85,B 0,C 180,E1 -18483.053,E2 -18483.053} C_VEL
LIN {X 0,Y 267.359,Z 279.658,A -85,B 0,C 180,E1 -18484.766,E2 -18484.766} C_VEL
LIN {X 0,Y 264.248,Z 274.302,A -85,B 0,C 180,E1 -18485.675,E2 -18485.675} C_VEL
LIN {X 0,Y 261.94,Z 270.317,A -85,B 0,C 180,E1 -18486.386,E2 -18486.386} C_VEL
LIN {X 0,Y 259.349,Z 265.83,A -85,B 0,C 180,E1 -18487.278,E2 -18487.278} C_VEL
LIN {X 0,Y 257.214,Z 258.919,A -85,B 0,C 180,E1 -18490.973,E2 -18490.973} C_VEL
LIN {X 0,Y 256.058,Z 255.135,A -85,B 0,C 180,E1 -18493.375,E2 -18493.375} C_VEL
LIN {X 0,Y 256.043,Z 255.086,A -85,B 0,C 180,E1 -18497.821,E2 -18497.821} C_VEL
LIN {X 0,Y 256.073,Z 255.081,A -85,B 0,C 180,E1 -18500.848,E2 -18500.848} C_VEL
LIN {X 0,Y 256.086,Z 255.084,A -85,B 0,C 180,E1 -18504.798,E2 -18504.798} C_VEL
LIN {X 0,Y 256.083,Z 255.088,A -85,B 0,C 180,E1 -18508.561,E2 -18508.561} C_VEL
LIN {X 0,Y 256.089,Z 255.086,A -85,B 0,C 180,E1 -18512.18,E2 -18512.18} C_VEL
LIN {X 0,Y 256.133,Z 255.08,A -85,B 0,C 180,E1 -18515.686,E2 -18515.686} C_VEL
LIN {X 0,Y 256.122,Z 255.083,A -85,B 0,C 180,E1 -18519.092,E2 -18519.092} C_VEL
LIN {X 0,Y 256.208,Z 255.062,A -85,B 0,C 180,E1 -18524.07,E2 -18524.07} C_VEL
LIN {X 0,Y 256.266,Z 255.059,A -85,B 0,C 180,E1 -18528.922,E2 -18528.922} C_VEL
LIN {X 0,Y 256.461,Z 255.035,A -85,B 0,C 180,E1 -18532.115,E2 -18532.115} C_VEL
LIN {X 0,Y 256.441,Z 255.036,A -85,B 0,C 180,E1 -18536.848,E2 -18536.848} C_VEL
LIN {X 0,Y 256.734,Z 254.999,A -85,B 0,C 180,E1 -18539.99,E2 -18539.99} C_VEL
LIN {X 0,Y 256.477,Z 255.034,A -85,B 0,C 180,E1 -18543.131,E2 -18543.131} C_VEL
LIN {X 0,Y 256.361,Z 255.242,A -85,B 0,C 180,E1 -18545.101,E2 -18545.101} C_VEL
LIN {X 0,Y 258.257,Z 260.855,A -85,B 0,C 180,E1 -18548.4,E2 -18548.4} C_VEL
LIN {X 0,Y 259.028,Z 262.531,A -85,B 0,C 180,E1 -18548.817,E2 -18548.817} C_VEL
LIN {X 0,Y 264.85,Z 271.821,A -85,B 0,C 180,E1 -18550.608,E2 -18550.608} C_VEL
LIN {X 0,Y 271.539,Z 283.667,A -85,B 0,C 180,E1 -18552.516,E2 -18552.516} C_VEL
LIN {X 0,Y 277.397,Z 295.893,A -85,B 0,C 180,E1 -18554.103,E2 -18554.103} C_VEL
LIN {X 0,Y 280.398,Z 303.707,A -85,B 0,C 180,E1 -18554.933,E2 -18554.933} C_VEL
LIN {X 0,Y 276.86,Z 369.819,A -85,B 0,C 180,E1 -18556.937,E2 -18556.937} C_VEL
LIN {X 0,Y 275.43,Z 383.521,A -85,B 0,C 180,E1 -18557.627,E2 -18557.627} C_VEL
LIN {X 0,Y 273.773,Z 395.655,A -85,B 0,C 180,E1 -18558.529,E2 -18558.529} C_VEL
LIN {X 0,Y 271.807,Z 406.803,A -85,B 0,C 180,E1 -18559.63,E2 -18559.63} C_VEL
LIN {X 0,Y 269.266,Z 418.853,A -85,B 0,C 180,E1 -18561.17,E2 -18561.17} C_VEL
LIN {X 0,Y 266.819,Z 428.909,A -85,B 0,C 180,E1 -18562.804,E2 -18562.804} C_VEL
LIN {X 0,Y 264.282,Z 438.163,A -85,B 0,C 180,E1 -18564.683,E2 -18564.683} C_VEL
LIN {X 0,Y 262.033,Z 446.088,A -85,B 0,C 180,E1 -18566.682,E2 -18566.682} C_VEL
LIN {X 0,Y 259.608,Z 453.909,A -85,B 0,C 180,E1 -18569.149,E2 -18569.149} C_VEL
LIN {X 0,Y 257.687,Z 460.023,A -85,B 0,C 180,E1 -18571.658,E2 -18571.658} C_VEL
LIN {X 0,Y 256.022,Z 465.318,A -85,B 0,C 180,E1 -18574.567,E2 -18574.567} C_VEL
LIN {X 0,Y 254.86,Z 468.862,A -85,B 0,C 180,E1 -18577.333,E2 -18577.333} C_VEL
LIN {X 0,Y 254.275,Z 470.639,A -85,B 0,C 180,E1 -18579.455,E2 -18579.455} C_VEL
LIN {X 0,Y 253.865,Z 471.717,A -85,B 0,C 180,E1 -18581.633,E2 -18581.633} C_VEL
LIN {X 0,Y 253.622,Z 472.041,A -85,B 0,C 180,E1 -18583.911,E2 -18583.911} C_VEL
LIN {X 0,Y 253.539,Z 471.544,A -85,B 0,C 180,E1 -18586.137,E2 -18586.137} C_VEL
LIN {X 0,Y 253.585,Z 470.173,A -85,B 0,C 180,E1 -18588.423,E2 -18588.423} C_VEL
LIN {X 0,Y 253.819,Z 467.813,A -85,B 0,C 180,E1 -18590.81,E2 -18590.81} C_VEL
LIN {X 0,Y 254.263,Z 464.332,A -85,B 0,C 180,E1 -18593.258,E2 -18593.258} C_VEL
LIN {X 0,Y 254.924,Z 459.524,A -85,B 0,C 180,E1 -18595.775,E2 -18595.775} C_VEL
LIN {X 0,Y 255.835,Z 453.063,A -85,B 0,C 180,E1 -18598.359,E2 -18598.359} C_VEL
LIN {X 0,Y 256.864,Z 446.342,A -85,B 0,C 180,E1 -18600.499,E2 -18600.499} C_VEL
LIN {X 0,Y 258.247,Z 437.608,A -85,B 0,C 180,E1 -18602.743,E2 -18602.743} C_VEL
LIN {X 0,Y 259.816,Z 427.666,A -85,B 0,C 180,E1 -18604.787,E2 -18604.787} C_VEL
LIN {X 0,Y 261.334,Z 417.659,A -85,B 0,C 180,E1 -18606.43,E2 -18606.43} C_VEL
LIN {X 0,Y 262.907,Z 405.462,A -85,B 0,C 180,E1 -18608.025,E2 -18608.025} C_VEL
LIN {X 0,Y 264.355,Z 392.854,A -85,B 0,C 180,E1 -18609.268,E2 -18609.268} C_VEL
LIN {X 0,Y 265.507,Z 379.528,A -85,B 0,C 180,E1 -18610.23,E2 -18610.23} C_VEL
LIN {X 0,Y 266.317,Z 366.931,A -85,B 0,C 180,E1 -18610.832,E2 -18610.832} C_VEL
LIN {X 0,Y 268.698,Z 298.807,A -85,B 0,C 180,E1 -18612.878,E2 -18612.878} C_VEL
LIN {X 0,Y 266.485,Z 286.557,A -85,B 0,C 180,E1 -18613.464,E2 -18613.464} C_VEL
LIN {X 0,Y 257.567,Z 261.582,A -85,B 0,C 180,E1 -18615.131,E2 -18615.131} C_VEL
LIN {X 0,Y 257.313,Z 260.536,A -85,B 0,C 180,E1 -18615.369,E2 -18615.369} C_VEL
LIN {X 0,Y 256.267,Z 255.104,A -85,B 0,C 180,E1 -18617.681,E2 -18617.681} C_VEL
